	(*
			[1] ETA_3111U1006XHE321XXXXXXZ01, ELT_Zaehler_BHKW_321_01
			Primaer-Adresse = 1
			Seriennummer = 3999427
			[2] ETA_3111U1006XHE322XXXXXXZ01, ELT_Zaehler_BHKW_322_01
			Primaer-Adresse = 2
			Seriennummer = 3999432
			[3] ETA_3111U1006BEST001XXXXXXZ01, ELT_Zaehler_Buerotrakt_01
			Primaer-Adresse = 3
			Seriennummer = 120267
			[4] ETA_3111U1006BEST002XXXXXXZ01, ELT_Zaehler_Gebaede_01
			Primaer-Adresse = 4
			Seriennummer = 205684
			[5] ETA_3111U1006BEST003XXXXXXZ01, ELT_Zaehler_Halle_TGA_01
			Primaer-Adresse = 5
			Seriennummer = 120264
			[6] ETA_3111EG005BEST004XXXXXXZ01, ELT_Zaehler_Halle_Licht_01
			Primaer-Adresse = 6
			Seriennummer = 214516
			[7] ETA_3111U1006BEST007XXXXXXZ01, GAS_Zaehler BHKW_007_01
			Primaer-Adresse = 7
			Seriennummer = 42078747
			[8] ETA_3111U1006BEST008XXXXXXZ01, GAS_Zaehler BHKW_008_01
			Primaer-Adresse = 8
			Seriennummer = 42078748
			[9] ETA_3111U1006BEST071XXXXXXZ01, WAERME_Zaehler WP_945_4371_01
			Primaer-Adresse = 71
			Seriennummer = 67694371
			[10] ETA_3111U1006BEST072XXXXXXZ01, WAERME_Zaehler WP_945_4372_01
			Primaer-Adresse = 72
			Seriennummer = 67694372
	*)
	Kommunikation_MBus	: ST_MBUS_Communication;
	Komm_MBus_WZaehler	: ST_MBUS_Communication;
	Komm_MBus_WZaehler2	: ST_MBUS_Communication;
	Komm_MBus_WZaehler_Basement	: ST_MBUS_Communication;

	aTelegramm_WMZ350 						: ARRAY[1..cMBUS_MaxTelegrams] OF ST_MBus_Data2;
	aTelegramm_WMZ305 						: ARRAY[1..cMBUS_MaxTelegrams] OF ST_MBus_Data2;
	aTelegramm_WMZ100 						: ARRAY[1..cMBUS_MaxTelegrams] OF ST_MBus_Data2;
	aTelegramm_WMZ300 						: ARRAY[1..cMBUS_MaxTelegrams] OF ST_MBus_Data2;
	aTelegramm_WMZ245 						: ARRAY[1..cMBUS_MaxTelegrams] OF ST_MBus_Data2;
	aTelegramm_WMZ235 						: ARRAY[1..cMBUS_MaxTelegrams] OF ST_MBus_Data2;
	aTelegramm_WMZ405 						: ARRAY[1..cMBUS_MaxTelegrams] OF ST_MBus_Data2;
	aTelegramm_WMZ425 						: ARRAY[1..cMBUS_MaxTelegrams] OF ST_MBus_Data2;
	aTelegramm_WMZ455 						: ARRAY[1..cMBUS_MaxTelegrams] OF ST_MBus_Data2;
	aTelegramm_WMZ342 						: ARRAY[1..cMBUS_MaxTelegrams] OF ST_MBus_Data2;
	
	
	aTelegramm_WMZ900 						: ARRAY[1..cMBUS_MaxTelegrams] OF ST_MBus_Data2;
	aTelegramm_WMZ935 						: ARRAY[1..cMBUS_MaxTelegrams] OF ST_MBus_Data2;
	
	aTelegramm_WMZ135						: ARRAY[1..cMBUS_MaxTelegrams] OF ST_MBus_Data2;
	aTelegramm_WMZ138						: ARRAY[1..cMBUS_MaxTelegrams] OF ST_MBus_Data2;
	aTelegramm_WMZ105						: ARRAY[1..cMBUS_MaxTelegrams] OF ST_MBus_Data2;
	aTelegramm_WMZ710						: ARRAY[1..cMBUS_MaxTelegrams] OF ST_MBus_Data2;
	aTelegramm_WMZ205						: ARRAY[1..cMBUS_MaxTelegrams] OF ST_MBus_Data2;
	aTelegramm_WMZ720						: ARRAY[1..cMBUS_MaxTelegrams] OF ST_MBus_Data2;
	
	Telegramm_WZ_Brennwerttherme			: ARRAY[1..cMBUS_MaxTelegrams] OF ST_MBus_Data2;
	Telegramm_WZ_BHKW_1						: ARRAY[1..cMBUS_MaxTelegrams] OF ST_MBus_Data2;
	Telegramm_WZ_BHKW_2						: ARRAY[1..cMBUS_MaxTelegrams] OF ST_MBus_Data2;
	Telegramm_WZ_Druckluftkompressor		: ARRAY[1..cMBUS_MaxTelegrams] OF ST_MBus_Data2;
	Telegramm_WZ_PWT_1						: ARRAY[1..cMBUS_MaxTelegrams] OF ST_MBus_Data2;
	Telegramm_WZ_Ofenkuehlung				: ARRAY[1..cMBUS_MaxTelegrams] OF ST_MBus_Data2;
	Telegramm_WZ_Abwaerme_Ofen_Abgasfackel	: ARRAY[1..cMBUS_MaxTelegrams] OF ST_MBus_Data2;
	Telegramm_GZ331_BWT	: ARRAY[1..cMBUS_MaxTelegrams] OF ST_MBus_Data2;


	Telegramm_SZ_BHKW_321		: ARRAY[1..cMBUS_MaxTelegrams] OF ST_MBus_Data2;
	Telegramm_SZ_BHKW_322		: ARRAY[1..cMBUS_MaxTelegrams] OF ST_MBus_Data2;
	Telegramm_SZ_Buerotrakt		: ARRAY[1..cMBUS_MaxTelegrams] OF ST_MBus_Data2;
	Telegramm_SZ_Gebaeude		: ARRAY[1..cMBUS_MaxTelegrams] OF ST_MBus_Data2;
	Telegramm_SZ_Halle_TGA		: ARRAY[1..cMBUS_MaxTelegrams] OF ST_MBus_Data2;
	Telegramm_SZ_Halle_Licht	: ARRAY[1..cMBUS_MaxTelegrams] OF ST_MBus_Data2;

	Telegramm_GZ_BHKW_321		: ARRAY[1..cMBUS_MaxTelegrams] OF ST_MBus_Data2;
	Telegramm_GZ_BHKW_322		: ARRAY[1..cMBUS_MaxTelegrams] OF ST_MBus_Data2;

	Telegramm_WZ_4371_WP_946	: ARRAY[1..cMBUS_MaxTelegrams] OF ST_MBus_Data2;
	Telegramm_WZ_4372_WP_946	: ARRAY[1..cMBUS_MaxTelegrams] OF ST_MBus_Data2;
	
	maxNumberOfNodes :INT := 22;
	cMSRLIBMaxNumberOfMBusDevices : BYTE := 18;	(*~
				Maximale Anzahl an MBus Geräten, die von der MSRlib unterstützt werden.
				Diese Konstante wird auch für die DP-Historisierung verwendet und muss grösser 6 (Anzahl der Basisdatentypen) sein.
				*)
	cMBUS_MaxData : INT := 40;
	(*cMBUS_MaxTelegrams : INT := 2;
	cMBUS_MaxCom : INT := 1;*)

END_VAR

// ---- POUs/MBUS_WZaehler.TcPOU
PROGRAM MBUS_WZaehler (* hier wird die Klemme, an welche der M-Bus mit den Zählern angeschlossen ist, alle 10ms aufgerufen *)
VAR
	Komm_Klemme_WZaehler		: FB_MBUSKL6781;
	Komm_Klemme_WZaehler2		: FB_MBUSKL6781;

	
	WMZ331_Brennwerttherme				: FB_MBUS_General_Ext;	(*1*)
	WMZ321_BHKW_1						: FB_MBUS_General_Ext;	(*3*)
	WMZ322_BHKW_2						: FB_MBUS_General_Ext;	(*4*)
	WMZ251_Druckluftkompressor			: FB_MBUS_General_Ext;	(*5*)
	WMZ215_PWT_1						: FB_MBUS_General_Ext;	(*6*)
	WMZ261_Ofenkuehlung_Dichtungen		: FB_MBUS_General_Ext;	(*7*)
	WMZ361_Abwaerme_Ofen_Abgasfackel	: FB_MBUS_General_Ext;	(*8*)

	adrBrennwerttherme				: ST_MBus_SecAdr := (udiIdNumber:=16#00474907);
	adrBHKW_1						: ST_MBus_SecAdr := (udiIdNumber:=16#00470996);
	adrBHKW_2						: ST_MBus_SecAdr := (udiIdNumber:=16#00474904);
	adrDruckluftkompressor			: ST_MBus_SecAdr := (udiIdNumber:=16#00552639);
	adrPWT_1						: ST_MBus_SecAdr := (udiIdNumber:=16#00455395);
	adrOfenkuehlung_Dichtungen		: ST_MBus_SecAdr := (udiIdNumber:=16#00482160);
	adrAbwaerme_Ofen_Abgasfackel	: ST_MBus_SecAdr := (udiIdNumber:=16#00482192);

	

	
END_VAR

Komm_Klemme_WZaehler(stComIn := IN_WZaehler, stComOut := OUT_WZaehler, stCom := Komm_MBus_WZaehler); // FB_MBUSKL6781
WMZ331_Brennwerttherme(usiAddress := 253, stSecAdr := adrBrennwerttherme, stCom := Komm_MBus_WZaehler); // FB_MBUS_General_Ext
Telegramm_WZ_Brennwerttherme := WMZ331_Brennwerttherme.arrTelegram;
WMZ321_BHKW_1(usiAddress := 253, stSecAdr := adrBHKW_1, stCom := Komm_MBus_WZaehler); // FB_MBUS_General_Ext
Telegramm_WZ_BHKW_1 := WMZ321_BHKW_1.arrTelegram;
WMZ322_BHKW_2(usiAddress := 253, stSecAdr := adrBHKW_2, stCom := Komm_MBus_WZaehler); // FB_MBUS_General_Ext
WMZ251_Druckluftkompressor(
    usiAddress := 253,
    stSecAdr := adrDruckluftkompressor,
    stCom := Komm_MBus_WZaehler); // FB_MBUS_General_Ext
WMZ215_PWT_1(usiAddress := 253, stSecAdr := adrPWT_1, stCom := Komm_MBus_WZaehler); // FB_MBUS_General_Ext
WMZ261_Ofenkuehlung_Dichtungen(
    usiAddress := 253,
    stSecAdr := adrOfenkuehlung_Dichtungen,
    stCom := Komm_MBus_WZaehler); // FB_MBUS_General_Ext
Telegramm_WZ_Ofenkuehlung := WMZ261_Ofenkuehlung_Dichtungen.arrTelegram;
WMZ361_Abwaerme_Ofen_Abgasfackel(
    usiAddress := 253,
    stSecAdr := adrAbwaerme_Ofen_Abgasfackel,
    stCom := Komm_MBus_WZaehler); // FB_MBUS_General_Ext
Telegramm_WZ_Abwaerme_Ofen_Abgasfackel := WMZ361_Abwaerme_Ofen_Abgasfackel.arrTelegram;
Telegramm_WZ_BHKW_2 := WMZ322_BHKW_2.arrTelegram;
Telegramm_WZ_Druckluftkompressor := WMZ251_Druckluftkompressor.arrTelegram;
Telegramm_WZ_PWT_1 := WMZ215_PWT_1.arrTelegram;

END_PROGRAM

// ---- POUs/MBUS_WZaehler2.TcPOU
PROGRAM MBUS_WZaehler2 (* hier wird die Klemme, an welche der M-Bus mit den Zählern angeschlossen ist, alle 10ms aufgerufen *)
VAR
	Komm_Klemme_WZaehler2		: FB_MBUSKL6781;
	WMZ135						: FB_MBUS_General_Ext;
	WMZ138						: FB_MBUS_General_Ext;
	WMZ105						: FB_MBUS_General_Ext;
	WMZ710						: FB_MBUS_General_Ext;
	WMZ205						: FB_MBUS_General_Ext;
	WMZ720						: FB_MBUS_General_Ext;

	adrWMZ135			: ST_MBus_SecAdr := (udiIdNumber:=16#13859504);
	adrWMZ138			: ST_MBus_SecAdr := (udiIdNumber:=16#13859500);
	adrWMZ105			: ST_MBus_SecAdr := (udiIdNumber:=16#12675097);
	adrWMZ205			: ST_MBus_SecAdr := (udiIdNumber:=16#13859501);
	adrWMZ710			: ST_MBus_SecAdr := (udiIdNumber:=16#12675093);
	adrWMZ720			: ST_MBus_SecAdr := (udiIdNumber:=16#13859505);
END_VAR

WMZ138(usiAddress := 253, stSecAdr := adrWMZ138, stCom := Komm_MBus_WZaehler2); // FB_MBUS_General_Ext
Komm_Klemme_WZaehler2(stComIn := IN_WZaehler2, stComOut := OUT_WZaehler2, stCom := Komm_MBus_WZaehler2); // FB_MBUSKL6781
aTelegramm_WMZ138 := WMZ138.arrTelegram;
WMZ135(usiAddress := 253, stSecAdr := adrWMZ135, stCom := Komm_MBus_WZaehler2); // FB_MBUS_General_Ext
aTelegramm_WMZ135 := WMZ135.arrTelegram;
WMZ105(usiAddress := 253, stSecAdr := adrWMZ105, stCom := Komm_MBus_WZaehler2); // FB_MBUS_General_Ext
WMZ205(usiAddress := 253, stSecAdr := adrWMZ205, stCom := Komm_MBus_WZaehler2); // FB_MBUS_General_Ext
aTelegramm_WMZ105 := WMZ105.arrTelegram;
aTelegramm_WMZ205 := WMZ205.arrTelegram;
WMZ710(usiAddress := 253, stSecAdr := adrWMZ710, stCom := Komm_MBus_WZaehler2); // FB_MBUS_General_Ext
aTelegramm_WMZ710 := WMZ710.arrTelegram;
WMZ720(usiAddress := 253, stSecAdr := adrWMZ720, stCom := Komm_MBus_WZaehler2); // FB_MBUS_General_Ext
aTelegramm_WMZ720 := WMZ720.arrTelegram;

END_PROGRAM

// ---- POUs/MBUS_WZaehler_Basement.TcPOU
PROGRAM MBUS_WZaehler_Basement (* hier wird die Klemme, an welche der M-Bus mit den Zählern angeschlossen ist, alle 10ms aufgerufen *)
VAR
	Komm_Klemme_WZaehler_Basement 		: FB_MBUSKL6781;

	WMZ350								: FB_MBUS_General_Ext;
	WMZ305								: FB_MBUS_General_Ext;
	WMZ300								: FB_MBUS_General_Ext;
	WMZ100								: FB_MBUS_General_Ext;
	WMZ455								: FB_MBUS_General_Ext;
	WMZ245								: FB_MBUS_General_Ext;
	WMZ235								: FB_MBUS_General_Ext;
	WMZ425								: FB_MBUS_General_Ext;
	WMZ900								: FB_MBUS_General_Ext;
	WMZ935								: FB_MBUS_General_Ext;
	WMZ342								: FB_MBUS_General_Ext;
	WMZ405								: FB_MBUS_General_Ext;
	
	//basement
	adrWMZ350					: ST_MBus_SecAdr := (udiIdNumber:=16#75372672);
	adrWMZ305					: ST_MBus_SecAdr := (udiIdNumber:=16#75234689);
	adrWMZ100					: ST_MBus_SecAdr := (udiIdNumber:=16#75494412);
	adrWMZ300					: ST_MBus_SecAdr := (udiIdNumber:=16#75878308);
	
	adrWMZ455					: ST_MBus_SecAdr := (udiIdNumber:=16#75375855);
	adrWMZ245					: ST_MBus_SecAdr := (udiIdNumber:=16#75563317);
	adrWMZ235					: ST_MBus_SecAdr := (udiIdNumber:=16#13859503);
	adrWMZ425					: ST_MBus_SecAdr := (udiIdNumber:=16#75878305);
	adrWMZ900					: ST_MBus_SecAdr := (udiIdNumber:=16#72925041);
	adrWMZ935					: ST_MBus_SecAdr := (udiIdNumber:=16#72925042);
	adrWMZ342					: ST_MBus_SecAdr := (udiIdNumber:=16#75375999);
	adrWMZ405					: ST_MBus_SecAdr := (udiIdNumber:=16#76089225);

END_VAR

Komm_Klemme_WZaehler_Basement(
    stComIn := IN_WZaehler_Basement,
    stComOut := OUT_WZaehler_Basement,
    stCom := Komm_MBus_WZaehler_Basement); // FB_MBUSKL6781
WMZ350(usiAddress := 253, stSecAdr := adrWMZ350, stCom := Komm_MBus_WZaehler_Basement); // FB_MBUS_General_Ext
aTelegramm_WMZ350 := WMZ350.arrTelegram;
WMZ305(usiAddress := 253, stSecAdr := adrWMZ305, stCom := Komm_MBus_WZaehler_Basement); // FB_MBUS_General_Ext
aTelegramm_WMZ305 := WMZ305.arrTelegram;
WMZ100(usiAddress := 253, stSecAdr := adrWMZ100, stCom := Komm_MBus_WZaehler_Basement); // FB_MBUS_General_Ext
WMZ300(usiAddress := 253, stSecAdr := adrWMZ300, stCom := Komm_MBus_WZaehler_Basement); // FB_MBUS_General_Ext
aTelegramm_WMZ100 := WMZ100.arrTelegram;
aTelegramm_WMZ300 := WMZ300.arrTelegram;
WMZ455(usiAddress := 253, stSecAdr := adrWMZ455, stCom := Komm_MBus_WZaehler_Basement); // FB_MBUS_General_Ext
aTelegramm_WMZ455 := WMZ455.arrTelegram;
WMZ245(usiAddress := 253, stSecAdr := adrWMZ245, stCom := Komm_MBus_WZaehler_Basement); // FB_MBUS_General_Ext
aTelegramm_WMZ245 := WMZ245.arrTelegram;
WMZ235(usiAddress := 253, stSecAdr := adrWMZ235, stCom := Komm_MBus_WZaehler_Basement); // FB_MBUS_General_Ext
aTelegramm_WMZ235 := WMZ235.arrTelegram;
WMZ425(usiAddress := 253, stSecAdr := adrWMZ425, stCom := Komm_MBus_WZaehler_Basement); // FB_MBUS_General_Ext
aTelegramm_WMZ425 := WMZ425.arrTelegram;
WMZ900(usiAddress := 253, stSecAdr := adrWMZ900, stCom := Komm_MBus_WZaehler_Basement); // FB_MBUS_General_Ext
aTelegramm_WMZ900 := WMZ900.arrTelegram;
WMZ935(usiAddress := 253, stSecAdr := adrWMZ935, stCom := Komm_MBus_WZaehler_Basement); // FB_MBUS_General_Ext
aTelegramm_WMZ935 := WMZ935.arrTelegram;
WMZ342(usiAddress := 253, stSecAdr := adrWMZ342, stCom := Komm_MBus_WZaehler_Basement); // FB_MBUS_General_Ext
aTelegramm_WMZ342 := WMZ342.arrTelegram;
WMZ405(usiAddress := 253, stSecAdr := adrWMZ405, stCom := Komm_MBus_WZaehler_Basement); // FB_MBUS_General_Ext
aTelegramm_WMZ405 := WMZ405.arrTelegram;

END_PROGRAM

// ---- POUs/MBUS_Zaehler.TcPOU
PROGRAM MBUS_Zaehler (* hier wird die Klemme, an welche der M-Bus mit den Zählern angeschlossen ist, alle 10ms aufgerufen *)
VAR
	Kommunikation_Klemme: FB_MBUSKL6781;

	Stromzaehler_BHKW_321		: FB_MBUS_General_Ext;
	Stromzaehler_BHKW_322	: FB_MBUS_General_Ext;
	Stromzaehler_Buerotrakt	: FB_MBUS_General_Ext;

	Stromzaehler_Gebaeude: FB_MBUS_General_Ext;
	Stromzaehler_Halle_TGA: FB_MBUS_General_Ext;
	Stromzaehler_Halle_Licht: FB_MBUS_General_Ext;
	Gaszaehler_BHKW1: FB_MBUS_General_Ext;
	Gaszaehler_BHKW2: FB_MBUS_General_Ext;

	WZ_4371_WP_946	: FB_MBUS_General_Ext;
	WZ_4372_WP_946	: FB_MBUS_General_Ext;
	
	
	
	
	
END_VAR

Kommunikation_Klemme(stComIn := IN_Stromzaehler, stComOut := OUT_Stromzaehler, stCom := Kommunikation_MBus); // FB_MBUSKL6781
Stromzaehler_BHKW_321(usiAddress := 1, stCom := Kommunikation_MBUS); // FB_MBUS_General_Ext
Telegramm_SZ_BHKW_321 := Stromzaehler_BHKW_321.arrTelegram;
Stromzaehler_BHKW_322(usiAddress := 2, stCom := Kommunikation_MBUS); // FB_MBUS_General_Ext
Telegramm_SZ_BHKW_322 := Stromzaehler_BHKW_322.arrTelegram;
Stromzaehler_Buerotrakt(usiAddress := 3, stCom := Kommunikation_MBUS); // FB_MBUS_General_Ext
Stromzaehler_Gebaeude(usiAddress := 4, stCom := Kommunikation_MBUS); // FB_MBUS_General_Ext
Stromzaehler_Halle_TGA(usiAddress := 5, stCom := Kommunikation_MBUS); // FB_MBUS_General_Ext
Stromzaehler_Halle_Licht(usiAddress := 6, stCom := Kommunikation_MBUS); // FB_MBUS_General_Ext
Telegramm_SZ_Halle_Licht := Stromzaehler_Halle_Licht.arrTelegram;
Gaszaehler_BHKW1(usiAddress := 7, stCom := Kommunikation_MBUS); // FB_MBUS_General_Ext
Telegramm_GZ_BHKW_321 := Gaszaehler_BHKW1.arrTelegram;
Gaszaehler_BHKW2(usiAddress := 8, stCom := Kommunikation_MBUS); // FB_MBUS_General_Ext
Telegramm_SZ_Buerotrakt := Stromzaehler_Buerotrakt.arrTelegram;
Telegramm_SZ_Gebaeude := Stromzaehler_Gebaeude.arrTelegram;
Telegramm_SZ_Halle_TGA := Stromzaehler_Halle_TGA.arrTelegram;
Telegramm_GZ_BHKW_322 := Gaszaehler_BHKW2.arrTelegram;
WZ_4371_WP_946(usiAddress := 71, stCom := Kommunikation_MBUS); // FB_MBUS_General_Ext
Telegramm_WZ_4371_WP_946 := WZ_4371_WP_946.arrTelegram;
WZ_4372_WP_946(usiAddress := 72, stCom := Kommunikation_MBUS); // FB_MBUS_General_Ext
Telegramm_WZ_4372_WP_946 := WZ_4372_WP_946.arrTelegram;

END_PROGRAM

// ---- POUs/MAIN.TcPOU
PROGRAM MAIN
VAR
	init_done		: BOOL := FALSE;
	
	//strategy controller
	Strategy : FB_StrategyController;
	//Strategy : FB_StrategyController_noChiller;
	//Strategy : FB_Strategycontroller_Conventional;
	//Strategy : FB_Strategycontroller_NoStorages;
	
	//thermal networks
	CN : FB_CoolingNetwork;
	HNLT_CN : FB_HnltCnLinkage;
	HNHT_CN : FB_HnhtCnLinkage;
	HNLT : FB_HeatingNetworkLowTemperature;
	HNHT_HNLT : FB_HnhtHnltLinkage;
	HNHT : FB_HeatingNetworkHighTemperature;

	
	//ambient state
	Ambient : FB_Ambient;
	
	//sensors
	LowVoltageMainDistribution : FB_LowVoltageMainDistribution;
END_VAR

//strategy controller
Strategy(ambientState := Ambient.localState,
	cnState := CN.localState,
	hnltState := HNLT.localState,
	hnhtState := HNHT.localState);

//ambient state
Ambient(sIPAddress := GlobalVariables.sIP_Ventilation);

//sensors
LowVoltageMainDistribution();
	
//thermal networks
CN(controlAutomatic := Strategy.cnControl);

HNLT_CN(controlAutomatic := Strategy.hnltCnLinkageControl,
	stAmbientState := Ambient.localState);
	
HNHT_CN(controlAutomatic := Strategy.hnhtCnLinkageControl);
	
HNLT(ambientState := Ambient.localState,
	controlAutomatic := Strategy.hnltControl);
	
HNHT_HNLT(controlAutomatic := Strategy.hnhtHnltLinkageControl);
	
HNHT(controlAutomatic := Strategy.hnhtControl,
	stAmbientState := Ambient.localState);
	


//Current implementation

(* --------------------------------------------------------------------------------------------------------------------------- *)

(* Analog- & Binaer Eingaenge - LESEN *)
(* P_Lesen; *)

	(* BUS Kommunikation - LESEN *)

(* --------------------------------------------------------------------------------------------------------------------------- *)
(* Starte Sub-Applikationen *)


	(*Initialisierung des Systems*)
	(*Einmalige Initialisierung der Parameter bei Hochlauf*)
	IF(NOT init_done) THEN
		Initialisierungsroutine();
		init_done := TRUE;
	END_IF;

	(* Allgemeine Parameter (Systemszeit, usw.) *)
	GA_Allgemein();

	(* Beleuchtung *)
	Beleuchtung();

END_PROGRAM

// ---- POUs/06 Strategy/FB_StrategyController.TcPOU
FUNCTION_BLOCK FB_StrategyController
VAR_INPUT
	ambientState : ST_AmbientState;
	
	//actual temperatures in thermal networks
	cnState : ST_ThermalNetworkState;
	hnltState : ST_ThermalNetworkState;
	hnhtState : ST_ThermalNetworkState;
END_VAR
VAR_OUTPUT	
	cnControl : ST_CoolingNetworkControl;
	hnltControl : ST_HeatingNetworkLowTemperatureControl;	
	hnhtControl : ST_HeatingNetworkHighTemperatureControl;
	hnltCnLinkageControl : ST_HnltCnLinkageControl;
	hnhtHnltLinkageControl : ST_HnhtHnltLinkageControl;
	hnhtCnLinkageControl : ST_HnhtCnLinkageControl;
END_VAR
VAR
	{attribute 'OPC.UA.DA' := '1'}
	localSetParameters : ST_StrategySetParameters;	
	{attribute 'OPC.UA.DA' := '1'}
	localState : ST_StrategyState;	

	//default parameters
	localDefaultParameters : ST_StrategyDefaultParameters;

	//internal variables
	fTargetTemperature_HNHT_Heating : REAL;
	fTargetTemperature_HNHT_Cooling : REAL;
	fTargetTemperature_HNLT_Cooling : REAL;
	fTargetTemperature_HNLT_Heating : REAL;
	fTargetTemperature_CN : REAL;
	aTemperatureLimits_HNHT : ARRAY[1..2] OF REAL;
	aTemperatureLimits_HNLT : ARRAY[1..2] OF REAL;
	aTemperatureLimits_CN : ARRAY[1..2] OF REAL;
	stHNHTCheckDefaultParameters : ST_RangeCheckDefaultParameters := (tTaskCycleTime := GlobalVariables.tCtrlCycleTime_MAIN, tCtrlCycleTime := GlobalVariables.tCtrlCycleTime_MAIN, fRestoreDifference := 5);
	HNHT_Check : FB_RangeCheck := (ST_DefaultParameters := stHNHTCheckDefaultParameters);
	stHNLTCheckDefaultParameters : ST_RangeCheckDefaultParameters := (tTaskCycleTime := GlobalVariables.tCtrlCycleTime_MAIN, tCtrlCycleTime := GlobalVariables.tCtrlCycleTime_MAIN, fRestoreDifference := 5);
	HNLT_Check : FB_RangeCheck := (ST_DefaultParameters := stHNLTCheckDefaultParameters);
	stCNCheckDefaultParameters : ST_RangeCheckDefaultParameters := (tTaskCycleTime := GlobalVariables.tCtrlCycleTime_MAIN, tCtrlCycleTime := GlobalVariables.tCtrlCycleTime_MAIN, fRestoreDifference := 2);
	CN_Check : FB_RangeCheck := (ST_DefaultParameters := stCNCheckDefaultParameters);
	
	
	//controller and variables for high temperature heating network
	fOffset_TargetTemperature_CHP1 : REAL; //not fixed, switches depending on ambient temperature -> see method: ControlHNHT
	fOffset_TargetTemperature_CHP2 : REAL; //not fixed, switches depending on ambient temperature -> see method: ControlHNHT
	fOffset_TargetTemperature_CondensingBoiler : REAL := 2;
	Controller_CHP_Prioritization : FB_CTRL_2POINT;
	Controller_CHP_Prioritization_Parameters : ST_CTRL_2POINT_PARAMS;	
	Controller_CHP1_UpperTemperature : FB_CTRL_2POINT; //check upper temperature for turning on chp
	Controller_CHP1_LowerTemperature : FB_CTRL_2POINT; //check lower temperature for turning off chp
	Controller_CHP1_Parameters : ST_CTRL_2POINT_PARAMS;	
	Trigger_CHP1_UpperTemperature : F_TRIG;
	Trigger_CHP1_LowerTemperature : F_TRIG;
	bTrigger_CHP1 : BOOL;
	Controller_CHP2_UpperTemperature : FB_CTRL_2POINT;
	Controller_CHP2_LowerTemperature : FB_CTRL_2POINT;
	Controller_CHP2_Parameters : ST_CTRL_2POINT_PARAMS;
	Trigger_CHP2_UpperTemperature : F_TRIG;
	Trigger_CHP2_LowerTemperature : F_TRIG;
	bTrigger_CHP2 : BOOL;
	Controller_CondensingBoiler : FB_CTRL_2POINT;
	Controller_CondensingBoiler_Parameters : ST_CTRL_2POINT_PARAMS;
	Controller_VSI_Loading_Permission : FB_CTRL_2POINT;
	Controller_VSI_Loading_Permission_Parameters : ST_CTRL_2POINT_PARAMS;
	Controller_VSI_Unloading_Permission : FB_CTRL_2POINT;
	Controller_VSI_Unloading_Permission_Parameters : ST_CTRL_2POINT_PARAMS;
	Controller_Buffer_VSI_Unloading : FB_CTRL_2POINT;
	Controller_Buffer_VSI_Unloading_Parameters : ST_CTRL_2POINT_PARAMS;
	Controller_StaticHeating : FB_CTRL_2POINT;
	Controller_StaticHeating_Parameters : ST_CTRL_2POINT_PARAMS;
	
	//controllers and variables for low temperature heating network
	Controller_OuterCapillaryTubeMats : FB_CTRL_2POINT;
	Controller_OuterCapillaryTubeMats_Parameters : ST_CTRL_2POINT_PARAMS;
	Controller_OuterCapillaryTubeMats_Permission : FB_CTRL_2POINT;
	Controller_OuterCapillaryTubeMats_Permission_Parameters : ST_CTRL_2POINT_PARAMS;
	fOffset_TargetTemperature_OuterCapillaryTubeMats_Cooling : REAL := 1;	
	fOffset_OuterCapillaryTubeMats_Permission : REAL := 10;
	
	Controller_HVFA_HNLT_HVFALoadingPermission : FB_CTRL_2POINT;
	Controller_HVFA_HNLT_HVFALoadingPermission_Parameters : ST_CTRL_2POINT_PARAMS;
	Controller_HVFA_HNLT_HVFAUnloadingPermission : FB_CTRL_2POINT;
	Controller_HVFA_HNLT_HVFAUnloadingPermission_Parameters : ST_CTRL_2POINT_PARAMS;
	Controller_Buffer_HVFA_HNLT_HVFAUnloading : FB_CTRL_2POINT;
	Controller_Buffer_HVFA_HNLT_HVFAUnloading_Parameters : ST_CTRL_2POINT_PARAMS;
	Controller_Buffer_HVFA_HNLT_HVFALoading : FB_CTRL_2POINT;
	Controller_Buffer_HVFA_HNLT_HVFALoading_Parameters : ST_CTRL_2POINT_PARAMS;
	Controller_HVFA_HNLT_Recooling : FB_CTRL_2POINT;
	Controller_HVFA_HNLT_Recooling_Parameters : ST_CTRL_2POINT_PARAMS;
	fOffset_TargetTemperature_HVFA_HNLT_Heating : REAL := 1;
	fOffset_HVFA_HNLT_Recooling : REAL := 16;
	fOffset_HVFA_HNLT_HVFALoadingPermission : REAL := 6;
	fOffset_Buffer_HVFA_HNLT_HVFALoading : REAL := 2;
		
	
	//controllers and variables for cooling network
	fOffset_TargetTemperature_eChiller : REAL := 2;	
	fOffset_TargetTemperature_HVFA_CN : REAL := 1;
	fOffset_TargetTemperature_HVFA_CN_Permission : REAL := 2.5;
	Controller_eChiller : FB_CTRL_2POINT;
	Controller_eChiller_Parameters : ST_CTRL_2POINT_PARAMS;	
	Controller_HVFA_CN_UnloadingPermission : FB_CTRL_2POINT;
	Controller_HVFA_CN_UnloadingPermission_Parameters : ST_CTRL_2POINT_PARAMS;
	Controller_Buffer_HVFA_CN_Unloading : FB_CTRL_2POINT;
	Controller_Buffer_HVFA_CN_Unloading_Parameters : ST_CTRL_2POINT_PARAMS;

	//controllers and variables for hnht and hnlt linkage
	Controller_HeatExchanger1 : FB_CTRL_2POINT;
	Controller_HeatExchanger1_Parameters : ST_CTRL_2POINT_PARAMS;
	fOffset_TargetTemperature_HeatExchanger1 : REAL := 2;
	Controller_HeatPump_HNHT : FB_CTRL_2POINT;
	Controller_HeatPump_HNHT_Parameters : ST_CTRL_2POINT_PARAMS;
	fOffset_TargetTemperature_HeatPump_HNHT : REAL := 3;
	Controller_HeatPump_HNLT : FB_CTRL_2POINT;
	Controller_HeatPump_HNLT_Parameters : ST_CTRL_2POINT_PARAMS;
	fOffset_TargetTemperature_HeatPump_HNHT_Permission : REAL := 4;
	
	//controllers and variables for hnlt and cn linkage
	fOffset_TargetTemperature_HeatPump : REAL;
	fOffset_TargetTemperature_HeatPump_Lower_CN_Permission : REAL;
	fOffset_TargetTemperature_HeatPump_Upper_CN_Permission : REAL;
	Controller_HeatPump : FB_CTRL_2POINT;
	Controller_HeatPump_Parameters : ST_CTRL_2POINT_PARAMS;
	Controller_HeatPump_Permission_Upper_CN : FB_CTRL_2POINT;
	Controller_HeatPump_Permission_Upper_CN_Parameters : ST_CTRL_2POINT_PARAMS;		
	Controller_HeatPump_Permission_Lower_CN : FB_CTRL_2POINT;
	Controller_HeatPump_Permission_Lower_CN_Parameters : ST_CTRL_2POINT_PARAMS;	

	//clock
	stDefaultParameters_Clock : ST_ClockDefaultParameters := (tTaskCycleTime := GlobalVariables.tCtrlCycleTime_MAIN, tCtrlCycleTime := T#1M);
	Clock : FB_Clock := (ST_DefaultParameters := stDefaultParameters_Clock);
END_VAR

Clock();
AmbientControl();
SetTemperatures();
ControlCN();
ControlHNLT();
ControlHNHT();
ControlHnltCnLinkage();
ControlHnhtHnltLinkage();
SetState();

METHOD AmbientControl : BOOL
VAR_INPUT
END_VAR
//check for heating or cooling mode
IF Clock.stClockState.sintMonth>4 AND Clock.stClockState.sintMonth<9 THEN
	//heating mode
	hnltCnLinkageControl.bHeatingMode := FALSE;
	hnhtCnLinkageControl.bHeatingMode := FALSE;
	localState.bHeatingMode := FALSE;
ELSE
	//cooling mode	
	hnltCnLinkageControl.bHeatingMode := TRUE;
	hnhtCnLinkageControl.bHeatingMode := TRUE;
	localState.bHeatingMode := TRUE;
END_IF
END_METHOD

METHOD ControlCN : BOOL
VAR_INPUT
END_VAR
//set hysteresis parameters for two-point controllers in cooling network
Controller_eChiller_Parameters.fHysteresisRange := 4;
Controller_eChiller_Parameters.tCtrlCycleTime := GlobalVariables.tCtrlCycleTime_MAIN;
Controller_eChiller_Parameters.tTaskCycleTime := GlobalVariables.tTaskCycleTime_MAIN;

//permission to unload storage depending on upper hvfa storage temperature
Controller_HVFA_CN_UnloadingPermission_Parameters.fHysteresisRange := 1;
Controller_HVFA_CN_UnloadingPermission_Parameters.tCtrlCycleTime := GlobalVariables.tCtrlCycleTime_MAIN;
Controller_HVFA_CN_UnloadingPermission_Parameters.tTaskCycleTime := GlobalVariables.tTaskCycleTime_MAIN;

//hysteresis for unloading hvfa storage depending on buffer storage temperature
Controller_Buffer_HVFA_CN_Unloading_Parameters.fHysteresisRange := 2;
Controller_Buffer_HVFA_CN_Unloading_Parameters.tCtrlCycleTime := GlobalVariables.tCtrlCycleTime_MAIN;
Controller_Buffer_HVFA_CN_Unloading_Parameters.tTaskCycleTime := GlobalVariables.tTaskCycleTime_MAIN;

//control eChiller
Controller_eChiller(fSetpointValue := cnState.fMidTemperature,
	fActualValue := fTargetTemperature_CN+fOffset_TargetTemperature_eChiller,
	eMode := eCTRL_MODE_ACTIVE,
	stParams := Controller_eChiller_Parameters);
	
//control hvfa storage unloading permission 
Controller_HVFA_CN_UnloadingPermission(fSetpointValue := fTargetTemperature_CN-fOffset_TargetTemperature_HVFA_CN_Permission,
	fActualValue := cnState.fLowerTemperature_ActiveStorage,
	eMode := eCTRL_MODE_ACTIVE,
	stParams := Controller_HVFA_CN_UnloadingPermission_Parameters);
	
//unloading permission buffer HVFA
Controller_Buffer_HVFA_CN_Unloading(fSetpointValue := cnState.fMidTemperature,
	fActualValue := fTargetTemperature_CN+fOffset_TargetTemperature_HVFA_CN,
	eMode := eCTRL_MODE_ACTIVE,
	stParams := Controller_Buffer_HVFA_CN_Unloading_Parameters);
	
//cnControl.bSetStatusOn_eChiller := Controller_eChiller.bOut;
//cnControl.bSetStatusOn_HVFASystem := (Controller_Buffer_HVFA_CN_Unloading.bOut AND Controller_HVFA_CN_UnloadingPermission.bOut) OR (hnltCnLinkageControl.bSetStatusOn_HeatPump AND NOT Controller_Buffer_HVFA_CN_Unloading.bOut AND NOT Controller_HVFA_CN_UnloadingPermission.bOut); 
//cnControl.bLoading_HVFASystem := NOT (Controller_Buffer_HVFA_CN_Unloading.bOut AND Controller_HVFA_CN_UnloadingPermission.bOut);

cnControl.bSetStatusOn_eChiller := TRUE;
cnControl.bSetStatusOn_HVFASystem := FALSE;
cnControl.bLoading_HVFASystem := FALSE;
END_METHOD

METHOD ControlHNHT : BOOL
VAR_INPUT
END_VAR
VAR
END_VAR
//set hysteresis parameters for two-point controllers in high temperature heating network
Controller_CHP_Prioritization_Parameters.fHysteresisRange := 4;
Controller_CHP_Prioritization_Parameters.tCtrlCycleTime := GlobalVariables.tCtrlCycleTime_MAIN;
Controller_CHP_Prioritization_Parameters.tTaskCycleTime := GlobalVariables.tTaskCycleTime_MAIN;

Controller_CHP1_Parameters.tCtrlCycleTime := GlobalVariables.tCtrlCycleTime_MAIN;
Controller_CHP1_Parameters.tTaskCycleTime := GlobalVariables.tTaskCycleTime_MAIN;
Controller_CHP2_Parameters.tCtrlCycleTime := GlobalVariables.tCtrlCycleTime_MAIN;
Controller_CHP2_Parameters.tTaskCycleTime := GlobalVariables.tTaskCycleTime_MAIN;

Controller_CondensingBoiler_Parameters.fHysteresisRange := 8;
Controller_CondensingBoiler_Parameters.tCtrlCycleTime := GlobalVariables.tCtrlCycleTime_MAIN;
Controller_CondensingBoiler_Parameters.tTaskCycleTime := GlobalVariables.tTaskCycleTime_MAIN;

Controller_Buffer_VSI_Unloading_Parameters.fHysteresisRange := 4;
Controller_Buffer_VSI_Unloading_Parameters.tCtrlCycleTime := GlobalVariables.tCtrlCycleTime_MAIN;
Controller_Buffer_VSI_Unloading_Parameters.tTaskCycleTime := GlobalVariables.tTaskCycleTime_MAIN;

Controller_VSI_Unloading_Permission_Parameters.fHysteresisRange := 4;
Controller_VSI_Unloading_Permission_Parameters.tCtrlCycleTime := GlobalVariables.tCtrlCycleTime_MAIN;
Controller_VSI_Unloading_Permission_Parameters.tTaskCycleTime := GlobalVariables.tTaskCycleTime_MAIN;

Controller_VSI_Loading_Permission_Parameters.fHysteresisRange := 4;
Controller_VSI_Loading_Permission_Parameters.tCtrlCycleTime := GlobalVariables.tCtrlCycleTime_MAIN;
Controller_VSI_Loading_Permission_Parameters.tTaskCycleTime := GlobalVariables.tTaskCycleTime_MAIN;

Controller_StaticHeating_Parameters.fHysteresisRange := 4;
Controller_StaticHeating_Parameters.tCtrlCycleTime := GlobalVariables.tCtrlCycleTime_MAIN;
Controller_StaticHeating_Parameters.tTaskCycleTime := GlobalVariables.tTaskCycleTime_MAIN;

Controller_CHP_Prioritization(fSetpointValue := 15,
	fActualValue := ambientState.fOutsideTemperature_Mean,
	eMode := eCTRL_MODE_ACTIVE,
	stParams := Controller_CHP_Prioritization_Parameters);
IF Controller_CHP_Prioritization.bOut THEN
	//prioritize large CHP (CHP2) during cold temperatures
	Controller_CHP1_Parameters.fHysteresisRange := 14;
	Controller_CHP2_Parameters.fHysteresisRange := 12;
	fOffset_TargetTemperature_CHP1 := 1;
	fOffset_TargetTemperature_CHP2 := 0;
ELSE
	//prioritize large CHP (CHP2) during cold temperatures
	Controller_CHP1_Parameters.fHysteresisRange := 12;
	Controller_CHP2_Parameters.fHysteresisRange := 14;	
	fOffset_TargetTemperature_CHP1 := 0;
	fOffset_TargetTemperature_CHP2 := 1;	
END_IF

//start when upper temperature too cold and stop when lower temperature too hot
Controller_CHP1_UpperTemperature(fSetpointValue := fTargetTemperature_HNHT_Heating-fOffset_TargetTemperature_CHP1,
	fActualValue := hnhtState.fUpperTemperature,
	eMode := eCTRL_MODE_ACTIVE,
	stParams := Controller_CHP1_Parameters);
Controller_CHP1_LowerTemperature(fSetpointValue := fTargetTemperature_HNHT_Heating-fOffset_TargetTemperature_CHP1,
	fActualValue := hnhtState.fLowerTemperature,
	eMode := eCTRL_MODE_ACTIVE,
	stParams := Controller_CHP1_Parameters);
Trigger_CHP1_UpperTemperature(CLK := Controller_CHP1_UpperTemperature.bOut);
Trigger_CHP1_LowerTemperature(CLK := Controller_CHP1_LowerTemperature.bOut);
IF Trigger_CHP1_UpperTemperature.Q THEN
	bTrigger_CHP1 := TRUE;
END_IF
IF Trigger_CHP1_LowerTemperature.Q THEN
	bTrigger_CHP1 := FALSE;
END_IF
hnhtControl.bSetStatusOn_CHP1 := Controller_CHP1_UpperTemperature.bOut OR (Controller_CHP1_LowerTemperature.bOut AND bTrigger_CHP1);

//start when upper temperature too cold and stop when lower temperature too hot
Controller_CHP2_UpperTemperature(fSetpointValue := fTargetTemperature_HNHT_Heating-fOffset_TargetTemperature_CHP2,
	fActualValue := hnhtState.fUpperTemperature,
	eMode := eCTRL_MODE_ACTIVE,
	stParams := Controller_CHP2_Parameters);
Controller_CHP2_LowerTemperature(fSetpointValue := fTargetTemperature_HNHT_Heating-fOffset_TargetTemperature_CHP2,
	fActualValue := hnhtState.fLowerTemperature,
	eMode := eCTRL_MODE_ACTIVE,
	stParams := Controller_CHP2_Parameters);
Trigger_CHP2_UpperTemperature(CLK := Controller_CHP2_UpperTemperature.bOut);
Trigger_CHP2_LowerTemperature(CLK := Controller_CHP2_LowerTemperature.bOut);
IF Trigger_CHP2_UpperTemperature.Q THEN
	bTrigger_CHP2 := TRUE;
END_IF
IF Trigger_CHP2_LowerTemperature.Q THEN
	bTrigger_CHP2 := FALSE;
END_IF
hnhtControl.bSetStatusOn_CHP2 := Controller_CHP2_UpperTemperature.bOut OR (Controller_CHP2_LowerTemperature.bOut AND bTrigger_CHP2);

Controller_CondensingBoiler(fSetpointValue := fTargetTemperature_HNHT_Heating-fOffset_TargetTemperature_CondensingBoiler,
	fActualValue := hnhtState.fMidTemperature,
	eMode := eCTRL_MODE_ACTIVE,
	stParams := Controller_CondensingBoiler_Parameters);
hnhtControl.bSetStatusOn_CondensingBoiler := Controller_CondensingBoiler.bOut;

//buffer storage asks VSI for unloading when buffer storage temperature falls below limit
Controller_Buffer_VSI_Unloading(fSetpointValue := fTargetTemperature_HNHT_Heating,
	fActualValue := hnhtState.fMidTemperature,
	eMode := eCTRL_MODE_ACTIVE,
	stParams := Controller_Buffer_VSI_Unloading_Parameters);

//VSI storage may only be unloaded when upper temperature is between limits for unloading
Controller_VSI_Unloading_Permission(fSetpointValue := hnhtState.fUpperTemperature_ActiveStorage,
	fActualValue := fTargetTemperature_HNHT_Heating,
	eMode := eCTRL_MODE_ACTIVE,
	stParams := Controller_VSI_Unloading_Permission_Parameters);
	
//VSI storage may only be loaded when lower temperature is between limits for loading
Controller_VSI_Loading_Permission(fSetpointValue := fTargetTemperature_HNHT_Heating,
	fActualValue := hnhtState.fLowerTemperature_ActiveStorage,
	eMode := eCTRL_MODE_ACTIVE,
	stParams := Controller_VSI_Loading_Permission_Parameters);
	
hnhtControl.bSetStatusOn_VSIStorage := (Controller_Buffer_VSI_Unloading.bOut AND Controller_VSI_Unloading_Permission.bOut AND NOT (hnhtControl.bSetStatusOn_CHP1 OR hnhtControl.bSetStatusOn_CHP2)) OR ((hnhtControl.bSetStatusOn_CHP1 OR hnhtControl.bSetStatusOn_CHP2) AND NOT Controller_Buffer_VSI_Unloading.bOut AND Controller_VSI_Loading_Permission.bOut); 
hnhtControl.bLoading_VSISystem := NOT Controller_Buffer_VSI_Unloading.bOut;

//condensing boiler is switched if network temperature falls below critical temperature limit
Controller_StaticHeating(fSetpointValue := 15,
	fActualValue := ambientState.fOutsideTemperature,
	eMode := eCTRL_MODE_ACTIVE,
	stParams := Controller_StaticHeating_Parameters);
hnhtControl.bSetStatusOn_StaticHeating := Controller_StaticHeating.bOut;
END_METHOD

METHOD ControlHnhtHnltLinkage : BOOL
VAR_INPUT
END_VAR
Controller_HeatExchanger1_Parameters.fHysteresisRange := 8;
Controller_HeatExchanger1_Parameters.tCtrlCycleTime := GlobalVariables.tCtrlCycleTime_MAIN;
Controller_HeatExchanger1_Parameters.tTaskCycleTime := GlobalVariables.tTaskCycleTime_MAIN;

Controller_HeatPump_HNHT_Parameters.fHysteresisRange := 4;
Controller_HeatPump_HNHT_Parameters.tCtrlCycleTime := GlobalVariables.tCtrlCycleTime_MAIN;
Controller_HeatPump_HNHT_Parameters.tTaskCycleTime := GlobalVariables.tTaskCycleTime_MAIN;

Controller_HeatPump_HNLT_Parameters.fHysteresisRange := 4;
Controller_HeatPump_HNLT_Parameters.tCtrlCycleTime := GlobalVariables.tCtrlCycleTime_MAIN;
Controller_HeatPump_HNLT_Parameters.tTaskCycleTime := GlobalVariables.tTaskCycleTime_MAIN;

//control heat exchanger 1
Controller_HeatExchanger1(fSetpointValue := fTargetTemperature_HNLT_Heating-fOffset_TargetTemperature_HeatExchanger1,
	fActualValue := hnltState.fMidTemperature,
	eMode := eCTRL_MODE_ACTIVE,
	stParams := Controller_HeatExchanger1_Parameters);
hnhtHnltLinkageControl.bSetStatusOn_HeatExchanger1 := Controller_HeatExchanger1.bOut;

//control heat pump hnht, return temperature HNHT should not exceed 60 °C
Controller_HeatPump_HNHT(fSetpointValue := fTargetTemperature_HNHT_Heating+fOffset_TargetTemperature_HeatPump_HNHT,
	fActualValue := hnhtState.fLowerTemperature,
	eMode := eCTRL_MODE_ACTIVE,
	stParams := Controller_HeatPump_HNHT_Parameters);
	
Controller_HeatPump_HNLT(fSetpointValue := hnltState.fMidTemperature,
	fActualValue := fTargetTemperature_HNLT_Cooling-fOffset_TargetTemperature_HeatPump_HNHT_Permission,
	eMode := eCTRL_MODE_ACTIVE,
	stParams := Controller_HeatPump_HNLT_Parameters);	
	
// If requested to cool HNLT and HNHT is not too hot, activate heat pump
hnhtHnltLinkageControl.bSetStatusOn_HeatPump := Controller_HeatPump_HNHT.bOut AND Controller_HeatPump_HNLT.bOut;
END_METHOD

METHOD ControlHNLT : BOOL
VAR_INPUT
END_VAR
//set hysteresis parameters for two-point controllers in cooling network
Controller_OuterCapillaryTubeMats_Parameters.fHysteresisRange := 6;
Controller_OuterCapillaryTubeMats_Parameters.tCtrlCycleTime := GlobalVariables.tCtrlCycleTime_MAIN;
Controller_OuterCapillaryTubeMats_Parameters.tTaskCycleTime := GlobalVariables.tTaskCycleTime_MAIN;

Controller_OuterCapillaryTubeMats_Permission_Parameters.fHysteresisRange := 6;
Controller_OuterCapillaryTubeMats_Permission_Parameters.tCtrlCycleTime := GlobalVariables.tCtrlCycleTime_MAIN;
Controller_OuterCapillaryTubeMats_Permission_Parameters.tTaskCycleTime := GlobalVariables.tTaskCycleTime_MAIN;


//control strategy for cooling network - fSetpointValue and fActualValue are changed for cooling applications
Controller_OuterCapillaryTubeMats(fSetpointValue := hnltState.fMidTemperature,
	fActualValue := fTargetTemperature_HNLT_Cooling+fOffset_TargetTemperature_OuterCapillaryTubeMats_Cooling,
	eMode := eCTRL_MODE_ACTIVE,
	stParams := Controller_OuterCapillaryTubeMats_Parameters);

//permission controller to ensure that network ist not heated up if ambient temperature is too high
Controller_OuterCapillaryTubeMats_Permission(fSetpointValue := fTargetTemperature_HNLT_Cooling-fOffset_OuterCapillaryTubeMats_Permission,
	fActualValue := ambientState.fOutsideTemperature,
	eMode := eCTRL_MODE_ACTIVE,
	stParams := Controller_OuterCapillaryTubeMats_Permission_Parameters);

//control hvfa storage
//set hysteresis parameters for two-point controllers in low temperature heating network

Controller_Buffer_HVFA_HNLT_HVFAUnloading_Parameters.fHysteresisRange := 2;
Controller_Buffer_HVFA_HNLT_HVFAUnloading_Parameters.tCtrlCycleTime := GlobalVariables.tCtrlCycleTime_MAIN;
Controller_Buffer_HVFA_HNLT_HVFAUnloading_Parameters.tTaskCycleTime := GlobalVariables.tTaskCycleTime_MAIN;

Controller_Buffer_HVFA_HNLT_HVFALoading_Parameters.fHysteresisRange := 4;
Controller_Buffer_HVFA_HNLT_HVFALoading_Parameters.tCtrlCycleTime := GlobalVariables.tCtrlCycleTime_MAIN;
Controller_Buffer_HVFA_HNLT_HVFALoading_Parameters.tTaskCycleTime := GlobalVariables.tTaskCycleTime_MAIN;

Controller_HVFA_HNLT_Recooling_Parameters.fHysteresisRange := 4;
Controller_HVFA_HNLT_Recooling_Parameters.tCtrlCycleTime := GlobalVariables.tCtrlCycleTime_MAIN;
Controller_HVFA_HNLT_Recooling_Parameters.tTaskCycleTime := GlobalVariables.tTaskCycleTime_MAIN;

Controller_HVFA_HNLT_HVFAUnloadingPermission_Parameters.fHysteresisRange := 4;
Controller_HVFA_HNLT_HVFAUnloadingPermission_Parameters.tCtrlCycleTime := GlobalVariables.tCtrlCycleTime_MAIN;
Controller_HVFA_HNLT_HVFAUnloadingPermission_Parameters.tTaskCycleTime := GlobalVariables.tTaskCycleTime_MAIN;

Controller_HVFA_HNLT_HVFALoadingPermission_Parameters.fHysteresisRange := 4;
Controller_HVFA_HNLT_HVFALoadingPermission_Parameters.tCtrlCycleTime := GlobalVariables.tCtrlCycleTime_MAIN;
Controller_HVFA_HNLT_HVFALoadingPermission_Parameters.tTaskCycleTime := GlobalVariables.tTaskCycleTime_MAIN;

//buffer storage asks HVFA_HNLT for unloading when buffer storage temperature falls below limit
Controller_Buffer_HVFA_HNLT_HVFAUnloading(fSetpointValue := fTargetTemperature_HNLT_Heating+fOffset_TargetTemperature_HVFA_HNLT_Heating,
	fActualValue := hnltState.fMidTemperature,
	eMode := eCTRL_MODE_ACTIVE,
	stParams := Controller_Buffer_HVFA_HNLT_HVFAUnloading_Parameters);
	
//buffer storage asks HVFA_HNLT for loading when buffer storage temperature rises above limit
Controller_Buffer_HVFA_HNLT_HVFALoading(fSetpointValue := hnltState.fMidTemperature,
	fActualValue := fTargetTemperature_HNLT_Cooling - fOffset_Buffer_HVFA_HNLT_HVFALoading,
	eMode := eCTRL_MODE_ACTIVE,
	stParams := Controller_Buffer_HVFA_HNLT_HVFALoading_Parameters);

//hvfa storage may only be unloaded when upper temperature is between limits for unloading
Controller_HVFA_HNLT_HVFAUnloadingPermission(fSetpointValue := hnltState.fLowerTemperature_ActiveStorage,
	fActualValue := fTargetTemperature_HNLT_Heating,
	eMode := eCTRL_MODE_ACTIVE,
	stParams := Controller_HVFA_HNLT_HVFAUnloadingPermission_Parameters);
	
//hvfa storage may only be loaded when lower temperature is between limits for loading
Controller_HVFA_HNLT_HVFALoadingPermission(fSetpointValue := fTargetTemperature_HNLT_Cooling - fOffset_HVFA_HNLT_HVFALoadingPermission,
	fActualValue := hnltState.fLowerTemperature_ActiveStorage,
	eMode := eCTRL_MODE_ACTIVE,
	stParams := Controller_HVFA_HNLT_HVFALoadingPermission_Parameters);

//enable hvfa recooling during low temperature times in summer months	
Controller_HVFA_HNLT_Recooling(fSetpointValue := hnltState.fLowerTemperature_ActiveStorage,
	fActualValue := fTargetTemperature_HNLT_Cooling-fOffset_HVFA_HNLT_Recooling,
	eMode := eCTRL_MODE_ACTIVE,
	stParams := Controller_HVFA_HNLT_Recooling_Parameters);
(*	
IF hnltCnLinkageControl.bHeatingMode THEN
	hnltControl.bSetStatusOn_HVFASystem := (Controller_HVFA_HNLT_HVFALoadingPermission.bOut AND Controller_Buffer_HVFA_HNLT_HVFALoading.bOut) OR (Controller_HVFA_HNLT_HVFAUnloadingPermission.bOut AND Controller_Buffer_HVFA_HNLT_HVFAUnloading.bOut);
	hnltControl.bLoading_HVFASystem := Controller_HVFA_HNLT_HVFALoadingPermission.bOut AND Controller_Buffer_HVFA_HNLT_HVFALoading.bOut;
	hnltControl.bSetStatusOn_OuterCapillaryTubeMats := Controller_OuterCapillaryTubeMats.bOut AND Controller_OuterCapillaryTubeMats_Permission.bOut;
ELSE
	hnltControl.bSetStatusOn_HVFASystem := ((Controller_HVFA_HNLT_HVFALoadingPermission.bOut AND Controller_Buffer_HVFA_HNLT_HVFALoading.bOut) OR (Controller_HVFA_HNLT_HVFAUnloadingPermission.bOut AND Controller_Buffer_HVFA_HNLT_HVFAUnloading.bOut)) OR (Controller_HVFA_HNLT_Recooling.bOut AND Controller_OuterCapillaryTubeMats_Permission.bOut);
	hnltControl.bLoading_HVFASystem := Controller_HVFA_HNLT_HVFALoadingPermission.bOut AND Controller_Buffer_HVFA_HNLT_HVFALoading.bOut;
	hnltControl.bSetStatusOn_OuterCapillaryTubeMats := (Controller_OuterCapillaryTubeMats.bOut AND Controller_OuterCapillaryTubeMats_Permission.bOut) OR (Controller_HVFA_HNLT_Recooling.bOut AND Controller_OuterCapillaryTubeMats_Permission.bOut);
END_IF
*)

IF Clock.stClockState.fHour > 6 AND Clock.stClockState.fHour < 22 THEN
	hnltControl.bSetStatusOn_HVFASystem := (Controller_HVFA_HNLT_HVFALoadingPermission.bOut AND Controller_Buffer_HVFA_HNLT_HVFALoading.bOut);
	hnltControl.bLoading_HVFASystem := Controller_HVFA_HNLT_HVFALoadingPermission.bOut AND Controller_Buffer_HVFA_HNLT_HVFALoading.bOut;
	hnltControl.bSetStatusOn_OuterCapillaryTubeMats := Controller_OuterCapillaryTubeMats.bOut;
ELSE
	hnltControl.bSetStatusOn_HVFASystem := Controller_HVFA_HNLT_Recooling.bOut ;
	hnltControl.bLoading_HVFASystem := FALSE;
	hnltControl.bSetStatusOn_OuterCapillaryTubeMats := Controller_HVFA_HNLT_Recooling.bOut OR Controller_OuterCapillaryTubeMats.bOut;
END_IF

// hnltControl.bSetStatusOn_OuterCapillaryTubeMats := Controller_OuterCapillaryTubeMats.bOut; AND Controller_OuterCapillaryTubeMats_Permission.bOut;
END_METHOD

METHOD ControlHnltCnLinkage : BOOL
VAR_INPUT
END_VAR
//set hysteresis parameters for hnlt cn linkage systems
fOffset_TargetTemperature_HeatPump := 0;
Controller_HeatPump_Parameters.fHysteresisRange := 4;
Controller_HeatPump_Parameters.tCtrlCycleTime := GlobalVariables.tCtrlCycleTime_MAIN;
Controller_HeatPump_Parameters.tTaskCycleTime := GlobalVariables.tTaskCycleTime_MAIN;

fOffset_TargetTemperature_HeatPump_Upper_CN_Permission := 4;
Controller_HeatPump_Permission_Upper_CN_Parameters.fHysteresisRange := 2;
Controller_HeatPump_Permission_Upper_CN_Parameters.tCtrlCycleTime := GlobalVariables.tCtrlCycleTime_MAIN;
Controller_HeatPump_Permission_Upper_CN_Parameters.tTaskCycleTime := GlobalVariables.tTaskCycleTime_MAIN;

fOffset_TargetTemperature_HeatPump_Lower_CN_Permission := 3;
Controller_HeatPump_Permission_Lower_CN_Parameters.fHysteresisRange := 4;
Controller_HeatPump_Permission_Lower_CN_Parameters.tCtrlCycleTime := GlobalVariables.tCtrlCycleTime_MAIN;
Controller_HeatPump_Permission_Lower_CN_Parameters.tTaskCycleTime := GlobalVariables.tTaskCycleTime_MAIN;
	
//control heat pump depending on heating demand in hnlt

Controller_HeatPump(fSetpointValue := fTargetTemperature_HNLT_Heating+fOffset_TargetTemperature_HeatPump,
	fActualValue := hnltState.fUpperTemperature,
	eMode := eCTRL_MODE_ACTIVE,
	stParams := Controller_HeatPump_Parameters);
	
Controller_HeatPump_Permission_Upper_CN(fSetpointValue := fTargetTemperature_CN+fOffset_TargetTemperature_HeatPump_Upper_CN_Permission,
	fActualValue := cnState.fUpperTemperature,
	eMode := eCTRL_MODE_ACTIVE,
	stParams := Controller_HeatPump_Permission_Lower_CN_Parameters);

Controller_HeatPump_Permission_Lower_CN(fSetpointValue := cnState.fMidTemperature,
	fActualValue := fTargetTemperature_CN-fOffset_TargetTemperature_HeatPump_Lower_CN_Permission,
	eMode := eCTRL_MODE_ACTIVE,
	stParams := Controller_HeatPump_Permission_Lower_CN_Parameters);
	
hnltCnLinkageControl.bSetStatusOn_HeatPump := Controller_HeatPump.bOut AND Controller_HeatPump_Permission_Lower_CN.bOut AND Controller_HeatPump_Permission_Upper_CN.bOut;
hnltCnLinkageControl.fTargetTemperature_ProductionHall := localDefaultParameters.fTargetTemperature_ProductionHall;

hnltCnLinkageControl.bSetStatusOn_InnerCapillaryTubeMats := TRUE;
hnltCnLinkageControl.bSetStatusOn_UnderfloorHeating := TRUE;
END_METHOD

METHOD SetState : BOOL
VAR_INPUT
END_VAR
localState.fTargetTemperature_HNHT_Heating := fTargetTemperature_HNHT_Heating;
localState.fTargetTemperature_HNHT_Cooling := fTargetTemperature_HNHT_Cooling;
localState.fTargetTemperature_HNLT_Heating := fTargetTemperature_HNLT_Heating;
localState.fTargetTemperature_HNLT_Cooling := fTargetTemperature_HNLT_Cooling;
localState.fTargetTemperature_CN := fTargetTemperature_CN;
localState.fTargetTemperature_ProductionHall := localDefaultParameters.fTargetTemperature_ProductionHall;

localState.aTemperatureLimits_HNHT := aTemperatureLimits_HNHT;
localState.aTemperatureLimits_HNLT := aTemperatureLimits_HNLT;
localState.aTemperatureLimits_CN := aTemperatureLimits_CN;
localState.bAlgorithmPermission_HNHT := HNHT_Check.bPermission;
localState.bAlgorithmPermission_HNLT := HNLT_Check.bPermission;
localState.bAlgorithmPermission_CN := CN_Check.bPermission;	

// localState.bHeatingMode state is set in AmbientControl

localState.fFeedTemperature_HNHT := fTargetTemperature_HNHT_Heating+localDefaultParameters.fOffset_FeedTemperature_HNHT;
localState.fFeedTemperature_HNLT_Heating := fTargetTemperature_HNLT_Heating+localDefaultParameters.fOffset_FeedTemperature_HNLT_Heating;
localState.fFeedTemperature_HNLT_Cooling := fTargetTemperature_HNLT_Cooling-localDefaultParameters.fOffset_FeedTemperature_HNLT_Cooling;
localState.fFeedTemperature_CN := fTargetTemperature_CN-localDefaultParameters.fOffset_FeedTemperature_CN;
END_METHOD

METHOD SetTemperatures : BOOL
VAR_INPUT
END_VAR
//set internal variables depending on prodution mode
IF localSetParameters.bProductionModeActivated THEN
	fTargetTemperature_CN := localDefaultParameters.fTargetTemperature_CN_ProductionMode;
	fTargetTemperature_HNLT_Heating := localDefaultParameters.fTargetTemperature_HNLT_Heating_ProductionMode;
	fTargetTemperature_HNLT_Cooling := localDefaultParameters.fTargetTemperature_HNLT_Cooling_ProductionMode;
	fTargetTemperature_HNHT_Heating := localDefaultParameters.fTargetTemperature_HNHT_Heating_ProductionMode;
	fTargetTemperature_HNHT_Cooling := localDefaultParameters.fTargetTemperature_HNHT_Cooling_ProductionMode;
	aTemperatureLimits_CN := localDefaultParameters.aTemperatureLimits_CN_ProductionMode;
	aTemperatureLimits_HNLT := localDefaultParameters.aTemperatureLimits_HNLT_ProductionMode;
	aTemperatureLimits_HNHT := localDefaultParameters.aTemperatureLimits_HNHT_ProductionMode;

ELSE
	fTargetTemperature_CN := localDefaultParameters.fTargetTemperature_CN;
	fTargetTemperature_HNLT_Heating := localDefaultParameters.fTargetTemperature_HNLT_Heating;
	fTargetTemperature_HNLT_Cooling := localDefaultParameters.fTargetTemperature_HNLT_Cooling;
	fTargetTemperature_HNHT_Heating := localDefaultParameters.fTargetTemperature_HNHT_Heating;
	fTargetTemperature_HNHT_Cooling := localDefaultParameters.fTargetTemperature_HNHT_Cooling;
	aTemperatureLimits_CN := localDefaultParameters.aTemperatureLimits_CN;
	aTemperatureLimits_HNLT := localDefaultParameters.aTemperatureLimits_HNLT;
	aTemperatureLimits_HNHT := localDefaultParameters.aTemperatureLimits_HNHT;
END_IF

//set feed temperatures
hnhtControl.fFeedTemperature := fTargetTemperature_HNHT_Heating+localDefaultParameters.fOffset_FeedTemperature_HNHT;
hnhtControl.fTargetTemperature := fTargetTemperature_HNHT_Heating;
hnltControl.fFeedTemperature_Heating := fTargetTemperature_HNLT_Heating+localDefaultParameters.fOffset_FeedTemperature_HNLT_Heating;
hnltControl.fFeedTemperature_Cooling := fTargetTemperature_HNLT_Cooling-localDefaultParameters.fOffset_FeedTemperature_HNLT_Cooling;
cnControl.fFeedTemperature := fTargetTemperature_CN-localDefaultParameters.fOffset_FeedTemperature_CN;
hnhtHnltLinkageControl.fFeedTemperature_HNHT := hnhtControl.fFeedTemperature;
hnhtHnltLinkageControl.fFeedTemperature_HNLT_Heating := hnltControl.fFeedTemperature_Heating;
hnhtHnltLinkageControl.fFeedTemperature_HNLT_Cooling := hnltControl.fFeedTemperature_Cooling;
hnltCnLinkageControl.fFeedTemperature_CN := cnControl.fFeedTemperature;
hnltCnLinkageControl.fFeedTemperature_HNLT_Heating := hnltControl.fFeedTemperature_Heating;
hnltCnLinkageControl.fFeedTemperature_HNLT_Cooling := hnltControl.fFeedTemperature_Cooling;

//set algorithm permission depending on production mode to control structs
CN_Check(fInput := cnState.fMidTemperature,
	fLowerLimit := aTemperatureLimits_CN[1],
	fUpperLimit := aTemperatureLimits_CN[2]);
cnControl.bAlgorithmPermission := CN_Check.bPermission;
	
HNLT_Check(fInput := hnltState.fMidTemperature,
	fLowerLimit := aTemperatureLimits_HNLT[1],
	fUpperLimit := aTemperatureLimits_HNLT[2]);
hnltControl.bAlgorithmPermission := HNLT_Check.bPermission;
	
HNHT_Check(fInput := hnhtState.fMidTemperature,
	fLowerLimit := aTemperatureLimits_HNHT[1],
	fUpperLimit := aTemperatureLimits_HNHT[2]);	
hnhtControl.bAlgorithmPermission := HNHT_Check.bPermission;
	
hnltCnLinkageControl.bAlgorithmPermission_CN := cnControl.bAlgorithmPermission;
hnltCnLinkageControl.bAlgorithmPermission_HNLT := hnltControl.bAlgorithmPermission;
hnhtHnltLinkageControl.bAlgorithmPermission_HNHT := hnhtControl.bAlgorithmPermission;
hnhtHnltLinkageControl.bAlgorithmPermission_HNLT := hnltControl.bAlgorithmPermission;
hnhtCnLinkageControl.bAlgorithmPermission_CN := cnControl.bAlgorithmPermission;
hnhtCnLinkageControl.bAlgorithmPermission_HNHT := hnhtControl.bAlgorithmPermission;
END_METHOD

END_FUNCTION_BLOCK

// ---- POUs/05 Thermal Networks/FB_CoolingNetwork.TcPOU
FUNCTION_BLOCK FB_CoolingNetwork
VAR_INPUT
	//control struct for cn
	controlAutomatic : ST_CoolingNetworkControl;	
END_VAR
VAR_OUTPUT
	{attribute 'OPC.UA.DA' := '1'}
	localState : ST_ThermalNetworkState;
END_VAR
VAR
	//systems
	BufferStorage : FB_BufferStorage;
	eChillerSystem : FB_eChillerSystem;
	HVFASystem : FB_HVFAStorageSystem;
	CentralMachineCoolingSystem : FB_CN_CentralMachineCooling;
	FlywheelMassStorageSystem : FB_FlywheelMassStorageSystem;
	
	//machines
	EMAG_GT : FB_EMAG_GT;
	EMAG_Y : FB_EMAG_Y;
	FlyhweelMassStorage : FB_FlywheelMassStorage;
	
	//internal variables
	bSetStatusOn_CentralMachineCooling : BOOL;
	bSetStatusOn_FlywheelMassStorage : BOOL;
END_VAR

//buffer storage system
BufferStorage();
localState.fUpperTemperature := BufferStorage.localState.fUpperTemperature;
localState.fMidTemperature := BufferStorage.localState.fMidTemperature;
localState.fLowerTemperature := BufferStorage.localState.fLowerTemperature;
localState.fUpperTemperature_ActiveStorage := HVFASystem.localStorageState.fUpperTemperature;
localState.fLowerTemperature_ActiveStorage := HVFASystem.localStorageState.fLowerTemperature;

//machines
EMAG_Y();
bSetStatusOn_CentralMachineCooling := EMAG_Y.bCN_Demand;

FlyhweelMassStorage();
bSetStatusOn_FlywheelMassStorage := FlyhweelMassStorage.bStatusOn;

//producer
eChillerSystem(bSetStatusOnAutomatic := controlAutomatic.bSetStatusOn_eChiller,
	bAlgorithmPermission := controlAutomatic.bAlgorithmPermission,
	fSetPointAutomatic := controlAutomatic.fFeedTemperature,
	fExternalTemperature := BufferStorage.localState.fMidTemperature,
	fReturnTemperature_Consumers := BufferStorage.localState.fUpperTemperature);

//consumer
//PU100 in central machine cooling system controls temperature difference of 3 K
CentralMachineCoolingSystem(bSetStatusOnAutomatic := bSetStatusOn_CentralMachineCooling,
	bAlgorithmPermission := controlAutomatic.bAlgorithmPermission,
	fSetPointAutomatic := 3); //temperature difference control

//PU191 in central machine cooling system controls return temperature of 20 degree
FlywheelMassStorageSystem(bSetStatusOnAutomatic := bSetStatusOn_FlywheelMassStorage,
	bAlgorithmPermission := controlAutomatic.bAlgorithmPermission,
	fSetPointAutomatic := 3); //temperature difference control
	
//external storages
HVFASystem(bSetStatusOnAutomatic := controlAutomatic.bSetStatusOn_HVFASystem,
	bAlgorithmPermission := controlAutomatic.bAlgorithmPermission,
	fSetPointAutomatic := 40,
	bLoadingAutomatic := controlAutomatic.bLoading_HVFASystem,
	aTelegramm_WMZ7x0 := aTelegramm_WMZ710,
	aTelegramm_WMZx05 := aTelegramm_WMZ105);

END_FUNCTION_BLOCK

// ---- POUs/03 Storages/FB_BufferStorage.TcPOU
FUNCTION_BLOCK FB_BufferStorage
VAR_INPUT
END_VAR
VAR_OUTPUT
	{attribute 'OPC.UA.DA' := '1'}	
	localState : ST_BufferStorageState;
END_VAR
VAR
	UpperTemperatureSensor : FB_TemperatureSensor; //upper temperature sensor
	MidTemperatureSensor : FB_TemperatureSensor; //mid temperature sensor
	LowerTemperatureSensor : FB_TemperatureSensor; //lower temperature sensor
	PressureSensor : FB_PressureSensor; //pressure sensor
END_VAR

//sensors
UpperTemperatureSensor();
MidTemperatureSensor();
LowerTemperatureSensor();
PressureSensor();

//get sensor inputs
UpperTemperatureSensor.GetState_AI();
MidTemperatureSensor.GetState_AI();
LowerTemperatureSensor.GetState_AI();
PressureSensor.GetState_AI();

//set outputs
localState.fUpperTemperature := UpperTemperatureSensor.fTemperature;
localState.fMidTemperature := MidTemperatureSensor.fTemperature;
localState.fLowerTemperature := LowerTemperatureSensor.fTemperature;

END_FUNCTION_BLOCK

// ---- POUs/04 Systems/CoolingSystems/FB_eChillerSystem.TcPOU
FUNCTION_BLOCK FB_eChillerSystem EXTENDS FB_SystemContinous
VAR_INPUT
	fExternalTemperature : REAL; //External temperature of buffer storage
	fReturnTemperature_Consumers : REAL;
END_VAR
VAR_OUTPUT
END_VAR
VAR
	//Efficient Energy eChiller 45-II
	eChiller : FB_eChiller;
	
	//discrete valve 138
	stSV138DefaultParameters : ST_MixingValveDefaultParameters := (fControllerAmplification := 1, tControllerIntegralTime := T#100S, fOutMinLimit := 30,  tTaskCycleTime := GlobalVariables.tTaskCycleTime_MAIN, tCtrlCycleTime := GlobalVariables.tCtrlCycleTime_MAIN,fOffsetTerminal := 3950);
	SV138 : FB_MixingValve := (ST_DefaultParameters := stSV138DefaultParameters); //valve motor needs continous signal but operates only between extreme positions	
	
	//heat counters
	stWMZ135DefaultParameters : ST_MollineC3HeatCounterDefaultParameters := (fSpecificHeatCapacity := 4.7);
	WMZ135 : FB_MollineC3HeatCounter := (ST_DefaultParameters := stWMZ135DefaultParameters);
	WMZ138 : FB_MollineC3HeatCounter;
	EM138 : FB_EmonioP3;
	
	//internal variables
	bSetStatusOn_eChiller : BOOL;
	bSetStatusOn_SV138 : BOOL;
END_VAR

MAIN();
eChiller.GetState();
eChiller(
	bSetStatusOnAutomatic := bSetStatusOn_eChiller,
	fSetPointAutomatic := fSetPoint,
	bAlgorithmPermission := bAlgorithmPermission,
	fExternalTemperature := fExternalTemperature,
	fReturnTemperature_Consumers := fReturnTemperature_Consumers);
eChiller.SetState();

SV138.GetState_AI();
SV138(
	bSetStatusOnAutomatic := bSetStatusOn_SV138,
	fSetPointAutomatic := 100,
	bAlgorithmPermission := bAlgorithmPermission,
	fThermalPowerExternal := WMZ138.fHeatFlowRate,
	nControlModeAutomatic := 0);
SV138.SetState_AO();

//insert heat counter telegramm from other task
WMZ135(aHeatCounterTelegramm := aTelegramm_WMZ135);
WMZ138(aHeatCounterTelegramm := aTelegramm_WMZ138);
EM138(sIPAddr := GlobalVariables.sIP_Emonio_eChiller);

METHOD PROTECTED  CheckError : BOOL
VAR_INPUT
END_VAR
VAR
	bError_eChiller : BOOL := FALSE;
	bError_SV138 : BOOL := FALSE;
END_VAR
VAR_OUTPUT
	bError : BOOL := FALSE;
END_VAR
//check chiller for error
bError_eChiller := eChiller.bError;

//check valve SV138 for error
IF SV138.fOperatingPoint < 95 AND eChiller.bStatusOn THEN
	bError_SV138 := TRUE;
END_IF

bError := bError_eChiller OR bError_SV138;
END_METHOD

METHOD PROTECTED  Operational : BOOL
VAR_INPUT
END_VAR
VAR_OUTPUT
	bSwitchToWorking : BOOL := FALSE;
END_VAR
bSetStatusOn_eChiller := TRUE;

IF eChiller.bStatusOn THEN
	bSwitchToWorking := TRUE;
END_IF
END_METHOD

METHOD PROTECTED  RampDown : BOOL
VAR_INPUT
END_VAR
VAR_OUTPUT
	bRampDownFinished : BOOL := FALSE;
END_VAR
bSetStatusOn_eChiller := FALSE;

//wait until eChiller is switched off before closing valve
IF NOT eChiller.bStatusOn THEN
	bSetStatusOn_SV138 := FALSE;
	IF SV138.fOperatingPoint < 20  THEN
		bRampDownFinished := TRUE;
	END_IF
END_IF
END_METHOD

METHOD PROTECTED  RampUp : BOOL
VAR_INPUT
END_VAR
VAR_OUTPUT
	bRampUpFinished : BOOL := FALSE;
END_VAR
bSetStatusOn_SV138 := TRUE;

//wait until valve is opened
IF SV138.fOperatingPoint > 85 THEN
	bRampUpFinished := TRUE;
END_IF
END_METHOD

METHOD PROTECTED   SetSetPointLimits : BOOL
VAR_INPUT
END_VAR
aSetPointLimits[1] := eChiller.ST_DefaultParameters.aSetPointLimitsTemperature[1];
aSetPointLimits[2] := eChiller.ST_DefaultParameters.aSetPointLimitsTemperature[2];
END_METHOD

METHOD PROTECTED  SetState : BOOL
VAR_INPUT
END_VAR
VAR_OUTPUT
END_VAR
fOperatingPoint := fExternalTemperature;

controlState.bStatusOn := bSetStatusOn;
setPointState.aSetPointLimits := aSetPointLimits;
setPointState.fSetPoint := fSetPoint;
setPointState.fOperatingPoint := fOperatingPoint;
setPointState.sSetPointUnit := 'degreeC';
setPointState.sOperatingPointUnit := 'degreeC';
END_METHOD

METHOD PROTECTED  Working : BOOL
VAR_INPUT
END_VAR
VAR_OUTPUT
	bSwitchToOperational : BOOL := FALSE;
END_VAR
//empty method
END_METHOD

END_FUNCTION_BLOCK

// ---- POUs/01 Actuators/CoolingUnits/FB_eChiller.TcPOU
FUNCTION_BLOCK FB_eChiller EXTENDS FB_ActuatorContinous
VAR_INPUT
	fExternalTemperature : REAL;
	fReturnTemperature_Consumers : REAL;
END_VAR
VAR_OUTPUT
	bError : BOOL;
END_VAR
VAR
	//default parameters
	localDefaultParameters : ST_eChillerDefaultParameters;

	{attribute 'OPC.UA.DA' := '1'}
	localState : ST_eChillerState;
	
	//analog converters
	OutputConverter_SetpointValue : FB_AnalogOutput(fUpperLimit := 60, fLowerLimit := -30);
	OutputConverter_ActualTemperature : FB_AnalogOutput(fUpperLimit := 60, fLowerLimit := -30);
	OutputConverter_ReturnTemperature_Consumers : FB_AnalogOutput(fUpperLimit := 60, fLowerLimit := -30);
	
	//I/O Links
	nSetPoint_OUT						AT %Q* : INT;
	nActualTemperature_OUT 				AT %Q* : INT; //Actual temperature in buffer storage linked to terminal
	nReturnTemperature_Consumers_OUT 	AT %Q* : INT;
	bSetStatusOn_OUT 					AT %Q* : BOOL;
	bError_IN 							AT %I* : BOOL;
	bWarning_IN 						AT %I* : BOOL;
	bStatusOn_IN 						AT %I* : BOOL;
END_VAR

MAIN();
OutputConverter_SetpointValue(fValue := fSetPoint);
OutputConverter_ActualTemperature(fValue := fExternalTemperature);
OutputConverter_ReturnTemperature_Consumers(fValue := fReturnTemperature_Consumers);

METHOD GetState : BOOL
VAR_INPUT
END_VAR
//control state
controlState.bStatusOn := bStatusOn_IN;
bStatusOn := bStatusOn_IN;

//setpoint state
setPointState.fOperatingPoint := fExternalTemperature;
setPointState.sOperatingPointUnit := 'degreeC';
fOperatingPoint := fExternalTemperature;

//local state
bError := bError_IN;
localState.bError := bError_IN;
localState.bWarning := bWarning_IN;
END_METHOD

METHOD PROTECTED  SetSetPointLimits : BOOL
VAR_INPUT
END_VAR
aSetPointLimits[1] := localDefaultParameters.aSetPointLimitsTemperature[1];
aSetPointLimits[2] := localDefaultParameters.aSetPointLimitsTemperature[2];
END_METHOD

METHOD SetState : BOOL
VAR_INPUT
END_VAR
//setpoint state
setPointState.fSetPoint := fSetPoint;
setPointState.sSetPointUnit := 'degreeC';
setPointState.aSetPointLimits := aSetPointLimits;

//outputs
nSetPoint_OUT := OutputConverter_SetpointValue.nValue;
nActualTemperature_OUT := OutputConverter_ActualTemperature.nValue;
nReturnTemperature_Consumers_OUT := OutputConverter_ReturnTemperature_Consumers.nValue;
bSetStatusOn_OUT := bSetStatusOn;
END_METHOD

PROPERTY ST_DefaultParameters : REFERENCE TO ST_eChillerDefaultParameters
GET
ST_DefaultParameters REF= localDefaultParameters;
END_GET
SET
localDefaultParameters := ST_DefaultParameters;
END_SET
END_PROPERTY

END_FUNCTION_BLOCK

// ---- POUs/04 Systems/StorageSystems/FB_HVFAStorageSystem.TcPOU
FUNCTION_BLOCK FB_HVFAStorageSystem EXTENDS FB_SystemContinous
VAR_INPUT
	bLoadingAutomatic : BOOL; //variable to determine if storage is in loading mode
	aTelegramm_WMZ7x0 : ARRAY[1..cMBUS_MaxTelegrams] OF ST_MBus_Data2;
	aTelegramm_WMZx05 : ARRAY[1..cMBUS_MaxTelegrams] OF ST_MBus_Data2;
END_VAR
VAR_OUTPUT	
	localStorageState : ST_HVFAStorageState;
END_VAR
VAR
	{attribute 'OPC.UA.DA' := '1'}
	localSetParameters : ST_ActiveStorageSystemSetParameters;
	{attribute 'OPC.UA.DA' := '1'}
	localState : ST_ActiveStorageSystemState;
	
	//default parameters
	localDefaultParameters : ST_HVFAStorageSystemDefaultParameters;	

	//storage
	HVFAStorage : FB_HVFAStorage;
	
	//pumps
	PUx05 : FB_PumpGrundfosMagna3; //Magna 3 pump (network side)
	PU7x0 : FB_Pump2Point; //CM pump (storage side)

	//valves
	stSVx05DefaultParameters : ST_MixingValveDefaultParameters := (tTaskCycleTime := GlobalVariables.tCtrlCycleTime_MAIN, tCtrlCycleTime := GlobalVariables.tCtrlCycleTime_MAIN, fOffsetTerminal := 3950);
	stSVx06DefaultParameters : ST_MixingValveDefaultParameters := (tTaskCycleTime := GlobalVariables.tCtrlCycleTime_MAIN, tCtrlCycleTime := GlobalVariables.tCtrlCycleTime_MAIN, fOffsetTerminal := 3950);
	stRVx05DefaultParameters : ST_MixingValveDefaultParameters := (tTaskCycleTime := GlobalVariables.tCtrlCycleTime_MAIN, tCtrlCycleTime := GlobalVariables.tCtrlCycleTime_MAIN, fOffsetTerminal := 3950, fControllerAmplification := 0.01);
	
	SVx05 : FB_MixingValve := (ST_DefaultParameters := stSVx05DefaultParameters); //discrete inlet valve, valve motor needs continous signal but operates only between extreme positions
	SVx06 : FB_MixingValve := (ST_DefaultParameters := stSVx06DefaultParameters); //discrete outlet valve	, valve motor needs continous signal but operates only between extreme positions
	RVx05 : FB_MixingValve := (ST_DefaultParameters := stRVx05DefaultParameters); //continous mixing valve
	
	//sensors
	WMZ7x0 : FB_MollineC3HeatCounter;
	WMZx05 : FB_MollineC3HeatCounter;
	
	//internal variables
	bSetStatusOn_PUx05 : BOOL;
	bSetStatusOn_PU7x0 : BOOL;
	bSetStatusOn_SVx05 : BOOL;
	fSetPoint_SVx05 : REAL;
	bSetStatusOn_SVx06 : BOOL;
	fSetPoint_SVx06 : REAL;	
	bSetStatusOn_RVx05 : BOOL;
	bLoading : BOOL;
	
	//triggers
	SwitchToLoading : R_TRIG;
	SwitchToUnloading : F_TRIG;
	bFinishedSwitchMode : BOOL := TRUE;
END_VAR

//storage
HVFAStorage(localState => localStorageState);

SelectLocalControlMode();
SwitchToLoading(CLK := bLoading);
SwitchToUnloading(CLK := bLoading);

//MAIN must be called before SwitchMode to prevent pump signal chattering (signal is written after SwitchMode function), SwitchMode may only be called if system is on
MAIN();

//disrupt calling SystemFlowControl via MAIN() when mode is switched and call SwitchMode()
IF ((SwitchToLoading.Q OR SwitchToUnloading.Q) OR NOT bFinishedSwitchMode) AND bSetStatusOn THEN
	SwitchMode(bSwitchToLoading := bLoading,
		bFinishedSwitchMode => bFinishedSwitchMode);
END_IF;

//pumps
PUx05.GetState_Profibus();
PUx05(bSetStatusOnAutomatic := bSetStatusOn_PUx05,
	fSetPointAutomatic := fSetPoint,
	bAlgorithmPermission := bAlgorithmPermission,
	nControlModeAutomatic := 0);
PUx05.SetState_Profibus();

PU7x0(bSetStatusOnAutomatic := bSetStatusOn_PU7x0,
	bAlgorithmPermission := bAlgorithmPermission);
PU7x0.SetState_BO();

//valves
SVx05.GetState_AI();
SVx05(bSetStatusOnAutomatic := bSetStatusOn_SVx05,
	fSetPointAutomatic := fSetPoint_SVx05,
	bAlgorithmPermission := bAlgorithmPermission,
	nControlModeAutomatic := 0);
SVx05.SetState_AO();

SVx06.GetState_AI();
SVx06(bSetStatusOnAutomatic := bSetStatusOn_SVx06,
	fSetPointAutomatic := fSetPoint_SVx06,
	bAlgorithmPermission := bAlgorithmPermission,
	nControlModeAutomatic := 0);
SVx06.SetState_AO();

//insert heat counter telegramm from other task
WMZ7x0(aHeatCounterTelegramm := aTelegramm_WMZ7x0);
WMZx05(aHeatCounterTelegramm := aTelegramm_WMZx05);

RVx05.GetState_AI();
RVx05(bSetStatusOnAutomatic := bSetStatusOn_RVx05,
	fSetPointAutomatic := 100,
	bAlgorithmPermission := bAlgorithmPermission,
	fThermalPowerExternal := WMZx05.fHeatFlowRate,
	nControlModeAutomatic := 0);
RVx05.SetState_AO();

METHOD PROTECTED  CheckError : BOOL
VAR_INPUT
END_VAR
VAR_OUTPUT
	bError : BOOL;
END_VAR
VAR
	bError_PUx05 : BOOL;
END_VAR
//check for pump error
bError_PUx05 := PUx05.bError;
END_METHOD

METHOD PROTECTED  Operational : BOOL
VAR_INPUT
END_VAR
VAR_OUTPUT
	bSwitchToWorking : BOOL := FALSE;
END_VAR
//storage pump
bSetStatusOn_PU7x0 := TRUE;

//network pump
bSetStatusOn_PUx05 := TRUE;

//temperature controlling valve
bSetStatusOn_RVx05 := TRUE;

IF PUx05.bStatusOn THEN
	bSwitchToWorking := TRUE;
END_IF
END_METHOD

METHOD PROTECTED  RampDown : BOOL
VAR_INPUT
END_VAR
VAR_OUTPUT
	bRampDownFinished : BOOL := FALSE;
END_VAR
bSetStatusOn_PU7x0 := FALSE;
bSetStatusOn_PUx05 := FALSE;
bSetStatusOn_RVx05 := FALSE;

IF RVx05.fOperatingPoint<20 AND NOT PUx05.bStatusOn THEN
	bRampDownFinished := TRUE;
END_IF
END_METHOD

METHOD PROTECTED  RampUp : BOOL
VAR_INPUT
END_VAR
VAR_OUTPUT
	bRampUpFinished : BOOL := FALSE;
END_VAR
bSetStatusOn_SVx05 := TRUE;
bSetStatusOn_SVx06 := TRUE;

IF bLoading = TRUE THEN
	fSetPoint_SVx05 := 0;
	fSetPoint_SVx06 := 0;
	IF SVx05.fOperatingPoint<20 AND SVx06.fOperatingPoint<20 THEN
		bRampUpFinished := TRUE;
	END_IF
ELSE
	fSetPoint_SVx05 := 100;
	fSetPoint_SVx06 := 100;
	IF SVx05.fOperatingPoint>80 AND SVx06.fOperatingPoint>80 THEN
		bRampUpFinished := TRUE;
	END_IF
END_IF
END_METHOD

METHOD PRIVATE SelectLocalControlMode : BOOL
VAR_INPUT
END_VAR
IF control.bManualModeActivated THEN
	bLoading := localSetParameters.bLoadingManual;
ELSIF control.bAlgorithmModeActivated AND bAlgorithmPermission THEN
	bLoading := localSetParameters.bLoadingAlgorithm;
ELSE
	bLoading := bLoadingAutomatic;
END_IF
END_METHOD

METHOD PROTECTED   SetSetPointLimits : BOOL
VAR_INPUT
END_VAR
aSetPointLimits[1] := localDefaultParameters.aSetPointLimitsTemperature[1];
aSetPointLimits[2] := localDefaultParameters.aSetPointLimitsTemperature[2];
END_METHOD

METHOD PROTECTED  SetState : BOOL
VAR_INPUT
END_VAR
VAR_OUTPUT
END_VAR
fOperatingPoint := PUx05.fOperatingPoint;

IF SVx05.fOperatingPoint<20 AND SVx06.fOperatingPoint<20 THEN
	localState.bLoading := TRUE;
ELSE
	localState.bLoading := FALSE;
END_IF

controlState.bStatusOn := bSetStatusOn;
setPointState.aSetPointLimits := aSetPointLimits;
setPointState.fSetPoint := fSetPoint;
setPointState.fOperatingPoint := fOperatingPoint;
setPointState.sSetPointUnit := 'percent';
setPointState.sOperatingPointUnit := 'percent';
END_METHOD

PROPERTY ST_DefaultParameters : REFERENCE TO ST_HVFAStorageSystemDefaultParameters
SET
localDefaultParameters := ST_DefaultParameters;
END_SET
END_PROPERTY

METHOD PRIVATE SwitchMode : BOOL
VAR_INPUT
	bSwitchToLoading : BOOL; //if false switch to cooling
END_VAR
VAR_OUTPUT
	bFinishedSwitchMode : BOOL := FALSE;
END_VAR
VAR_INST
	bRampDownFinished : BOOL := FALSE;
END_VAR
//check system state
IF bRampDownFinished THEN
	IF bSwitchToLoading THEN
		fSetPoint_SVx05 := 0;
		fSetPoint_SVx06 := 0;
		IF SVx05.fOperatingPoint<20 AND SVx06.fOperatingPoint<20 THEN
			//reset instant variable and switch on pump
			bRampDownFinished := FALSE;			
			bFinishedSwitchMode := TRUE;
			bSetStatusOn_PUx05 := TRUE;
		END_IF
		
	ELSE
		fSetPoint_SVx05 := 100;
		fSetPoint_SVx06 := 100;
		IF SVx05.fOperatingPoint>80 AND SVx06.fOperatingPoint>80 THEN
			//reset instant variable and switch on pump
			bRampDownFinished := FALSE;			
			bFinishedSwitchMode := TRUE;
			bSetStatusOn_PUx05 := TRUE;
		END_IF
	END_IF
ELSE
	bSetStatusOn_PUx05 := FALSE;
	IF NOT PUx05.bStatusOn THEN
		bRampDownFinished := TRUE;
	END_IF
END_IF
END_METHOD

METHOD PROTECTED  Working : BOOL
VAR_INPUT
END_VAR
VAR_OUTPUT
	bSwitchToOperational : BOOL := FALSE;
END_VAR
//empty method
END_METHOD

END_FUNCTION_BLOCK

// ---- POUs/03 Storages/FB_HVFAStorage.TcPOU
FUNCTION_BLOCK FB_HVFAStorage
VAR_INPUT
END_VAR
VAR_OUTPUT
	{attribute 'OPC.UA.DA' := '1'}
	localState : ST_HVFAStorageState;
END_VAR
VAR
	UpperTemperatureSensor : FB_TemperatureSensor; //upper temperature sensor
	LowerTemperatureSensor : FB_TemperatureSensor; //lower temperature sensor
END_VAR

//get sensor inputs
UpperTemperatureSensor.GetState_AI();
LowerTemperatureSensor.GetState_AI();

//set outputs
localState.fUpperTemperature := UpperTemperatureSensor.fTemperature;
localState.fLowerTemperature := LowerTemperatureSensor.fTemperature;

END_FUNCTION_BLOCK

// ---- POUs/01 Actuators/Pumps/FB_Pump2Point.TcPOU
FUNCTION_BLOCK FB_Pump2Point EXTENDS FB_Actuator2Point
VAR
	//I/O Links
	bSetStatusOn_OUT 	AT %Q* : BOOL := FALSE;
END_VAR

SelectControlMode();

METHOD SetState_BO : BOOL
VAR_INPUT
END_VAR
//output
bSetStatusOn_OUT := bSetStatusOn;
END_METHOD

END_FUNCTION_BLOCK

// ---- POUs/04 Systems/ConsumerSystems/CN/FB_CN_CentralMachineCooling.TcPOU
FUNCTION_BLOCK FB_CN_CentralMachineCooling EXTENDS FB_SystemContinous
VAR_INPUT
END_VAR
VAR_OUTPUT
END_VAR
VAR
	//default parameters
	localDefaultParameters : ST_CN_CentralMachineCoolingDefaultParameters;
	
	//pumps
	stPU100DefaultParameters : ST_PumpGrundfosMagna3DefaultParameters := (tTaskCycleTime := GlobalVariables.tTaskCycleTime_MAIN, tCtrlCycleTime := GlobalVariables.tCtrlCycleTime_MAIN);
	PU100 : FB_PumpGrundfosMagna3 := (ST_DefaultParameters := stPU100DefaultParameters);;

	//valves
	stSV100DefaultParameters : ST_DiscreteValveDefaultParameters := (nFeedback := 3);
	SV100 : FB_DiscreteValve := (ST_DefaultParameters := stSV100DefaultParameters);
	
	//heat counters
	WMZ100: FB_MollineEHeatCounter;
	
	//internal variables
	bSetStatusOn_PU100 : BOOL;
	bSetStatusOn_SV100 : BOOL;
END_VAR

MAIN();

SV100.GetState_BI();
SV100(bSetStatusOnAutomatic := bSetStatusOn_SV100,
	bAlgorithmPermission := bAlgorithmPermission);
SV100.SetState_BO();

PU100.GetState_Profibus();
PU100(bSetStatusOnAutomatic := bSetStatusOn_PU100,
	bAlgorithmPermission := bAlgorithmPermission,
	fSetPointAutomatic := fSetPoint,
	nControlModeAutomatic := 3,
	fThermalPowerExternal := WMZ100.fHeatFlowRate);
PU100.SetState_Profibus();

WMZ100(aHeatCounterTelegramm:=aTelegramm_WMZ100);

METHOD PROTECTED  CheckError : BOOL
VAR_INPUT
END_VAR
VAR_OUTPUT
	bError : BOOL;
END_VAR
IF (PU100.bStatusOn AND SV100.localState.nPosition = 2) OR PU100.bError THEN
	bError := TRUE;
END_IF
END_METHOD

METHOD PROTECTED  Operational : BOOL
VAR_INPUT
END_VAR
VAR_OUTPUT
	bSwitchToWorking : BOOL := FALSE;
END_VAR
bSetStatusOn_PU100 := TRUE;

IF PU100.bStatusOn THEN
	bSwitchToWorking := TRUE;
END_IF
END_METHOD

METHOD PROTECTED  RampDown : BOOL
VAR_INPUT
END_VAR
VAR_OUTPUT
	bRampDownFinished : BOOL := FALSE;
END_VAR
bSetStatusOn_PU100 := FALSE;

IF NOT PU100.bStatusOn THEN
	bSetStatusOn_SV100 := FALSE;
	IF SV100.localState.nPosition = 2 THEN
		bRampDownFinished := TRUE;
	END_IF
END_IF
END_METHOD

METHOD PROTECTED  RampUp : BOOL
VAR_INPUT
END_VAR
VAR_OUTPUT
	bRampUpFinished : BOOL := FALSE;
END_VAR
bSetStatusOn_SV100 := TRUE;

IF SV100.localState.nPosition = 3 THEN
	bRampUpFinished := TRUE;
END_IF
END_METHOD

METHOD PROTECTED   SetSetPointLimits : BOOL
VAR_INPUT
END_VAR
IF  PU100.nControlModeAutomatic = 3 THEN
	aSetPointLimits[1] := localDefaultParameters.aSetPointLimitsTemperatureDifference[1];
	aSetPointLimits[2] := localDefaultParameters.aSetPointLimitsTemperatureDifference[2];
ELSE
	aSetPointLimits[1] := localDefaultParameters.aSetPointLimitsRelativeSpeed[1];
	aSetPointLimits[2] := localDefaultParameters.aSetPointLimitsRelativeSpeed[2];
END_IF
END_METHOD

METHOD PROTECTED  SetState : BOOL
VAR_INPUT
END_VAR
VAR_OUTPUT
END_VAR
fOperatingPoint := PU100.localState.fTemperatureDifference;

controlState.bStatusOn := bSetStatusOn;
setPointState.aSetPointLimits := aSetPointLimits;
setPointState.fSetPoint := fSetPoint;
setPointState.fOperatingPoint := fOperatingPoint;
setPointState.sSetPointUnit := 'K';
setPointState.sOperatingPointUnit := 'K';
END_METHOD

METHOD PROTECTED  Working : BOOL
VAR_INPUT
END_VAR
VAR_OUTPUT
	bSwitchToOperational : BOOL := FALSE;
END_VAR
//empty method
END_METHOD

END_FUNCTION_BLOCK

// ---- POUs/04 Systems/ConsumerSystems/CN/FB_FlywheelMassStorageSystem.TcPOU
FUNCTION_BLOCK FB_FlywheelMassStorageSystem EXTENDS FB_SystemContinous
VAR_INPUT
END_VAR
VAR_OUTPUT
END_VAR
VAR
	//default parameters
	localDefaultParameters : ST_FlywheelMassStorageDefaultParameters;	

	//pumps
	stPU191DefaultParameters : ST_PumpGrundfosMagna3DefaultParameters := (tTaskCycleTime := GlobalVariables.tTaskCycleTime_MAIN, tCtrlCycleTime := GlobalVariables.tCtrlCycleTime_MAIN);
	PU191 : FB_PumpGrundfosMagna3 := (ST_DefaultParameters := stPU191DefaultParameters);;

	//valves
	stSV191DefaultParameters : ST_DiscreteValveDefaultParameters := (nFeedback := 0);
	SV191 : FB_DiscreteValve := (ST_DefaultParameters := stSV191DefaultParameters);
	
	//internal variables
	bSetStatusOn_PU191 : BOOL;
	bSetStatusOn_SV191 : BOOL;
	
	bStartTimer : BOOL;
	Timer : TON;
END_VAR

MAIN();

//use timer because valve has no feedback signal
Timer(IN := bStartTimer,
	PT := T#75S);

SV191.GetState_BI();
SV191(bSetStatusOnAutomatic := bSetStatusOn_SV191,
	bAlgorithmPermission := bAlgorithmPermission);
SV191.SetState_BO();

//pump controls return temperature
PU191.GetState_Profibus();
PU191(bSetStatusOnAutomatic := bSetStatusOn_PU191,
	bAlgorithmPermission := bAlgorithmPermission,
	fSetPointAutomatic := fSetPoint,
	nControlModeAutomatic := 3);
PU191.SetState_Profibus();

METHOD PROTECTED  CheckError : BOOL
VAR_INPUT
END_VAR
VAR_OUTPUT
	bError : BOOL;
END_VAR
bError := PU191.bError;
END_METHOD

METHOD PROTECTED  Operational : BOOL
VAR_INPUT
END_VAR
VAR_OUTPUT
	bSwitchToWorking : BOOL := FALSE;
END_VAR
bSetStatusOn_PU191 := TRUE;

IF PU191.bStatusOn THEN
	bSwitchToWorking := TRUE;
END_IF
END_METHOD

METHOD PROTECTED  RampDown : BOOL
VAR_INPUT
END_VAR
VAR_OUTPUT
	bRampDownFinished : BOOL := FALSE;
END_VAR
bSetStatusOn_PU191 := FALSE;

IF NOT PU191.bStatusOn THEN
	bSetStatusOn_SV191 := FALSE;
	bStartTimer := TRUE;
	IF Timer.Q THEN
		bStartTimer := FALSE;
		bRampDownFinished := TRUE;
	END_IF
END_IF
END_METHOD

METHOD PROTECTED  RampUp : BOOL
VAR_INPUT
END_VAR
VAR_OUTPUT
	bRampUpFinished : BOOL := FALSE;
END_VAR
bSetStatusOn_SV191 := TRUE;
bStartTimer := TRUE;

IF Timer.Q THEN
	bStartTimer := FALSE;
	bRampUpFinished := TRUE;
END_IF
END_METHOD

METHOD PROTECTED   SetSetPointLimits : BOOL
VAR_INPUT
END_VAR
IF  PU191.nControlModeAutomatic = 3 THEN
	aSetPointLimits[1] := localDefaultParameters.aSetPointLimitsTemperatureDifference[1];
	aSetPointLimits[2] := localDefaultParameters.aSetPointLimitsTemperatureDifference[2];
ELSE
	aSetPointLimits[1] := localDefaultParameters.aSetPointLimitsRelativeSpeed[1];
	aSetPointLimits[2] := localDefaultParameters.aSetPointLimitsRelativeSpeed[2];
END_IF
END_METHOD

METHOD PROTECTED  SetState : BOOL
VAR_INPUT
END_VAR
VAR_OUTPUT
END_VAR
fOperatingPoint := PU191.localState.fTemperatureDifference;

controlState.bStatusOn := bSetStatusOn;
setPointState.aSetPointLimits := aSetPointLimits;
setPointState.fSetPoint := fSetPoint;
setPointState.fOperatingPoint := fOperatingPoint;
setPointState.sSetPointUnit := 'K';
setPointState.sOperatingPointUnit := 'K';
END_METHOD

METHOD PROTECTED  Working : BOOL
VAR_INPUT
END_VAR
VAR_OUTPUT
	bSwitchToOperational : BOOL := FALSE;
END_VAR
//empty method
END_METHOD

END_FUNCTION_BLOCK

// ---- POUs/01 Actuators/ConsumerUnits/FB_EMAG_GT.TcPOU
FUNCTION_BLOCK FB_EMAG_GT
VAR_INPUT
END_VAR
VAR_OUTPUT
	bStatusOn : BOOL;
	bError_Connection : BOOL;
END_VAR
VAR
	OPC_UA				: FB_OPC_UA_READ;
	stOPC_UA_Server		: ST_OPC_UA_Server;
	sOPC_UA_Server_URL 	: STRING;
	sNamespaceName		: STRING;
	aNodes				: ARRAY[1..2] OF ST_OPC_UANode;
	nNodeCount			: UDINT := 2;
	stIndexRange		: ARRAY [1..nMaxIndexRange] OF ST_UAIndexRange;
	currentNode			: UDINT := 1;
	
	bStatusOn_CoolingLubricant : BOOL;
	bStatusOn_Machine : BOOL;
	
	// timer
	bStartTimer : BOOL;
	Timer : TON;
END_VAR

sOPC_UA_Server_URL 	:= GlobalVariables.sIP_EMAG_GT;
sNamespaceName 		:= 'http://www.boschrexroth.com/IndraLogic';

(*Define Nodes to Read*)
aNodes[1].NodeID.sIdentifier			:= 'Application.Kuehlung_Anforderung.Kuehlung_KSS_blau_ON';
aNodes[1].NodeID.eIdentifierType		:= eUAIdentifierType_String;
aNodes[1].SizeOfDataType				:= DINT_TO_UDINT(eUAType_Boolean);
aNodes[1].NodeAddInfo.nIndexRangeCount 	:= 0;
aNodes[1].NodeAddInfo.stIndexRange		:= stIndexRange;
aNodes[1].TargetVar						:= ADR(bStatusOn_CoolingLubricant);

aNodes[2].NodeID.sIdentifier			:= 'Application.Kuehlung_Anforderung.Kuehlung_Maschine_blau_ON';
aNodes[2].NodeID.eIdentifierType		:= eUAIdentifierType_String;
aNodes[2].SizeOfDataType				:= DINT_TO_UDINT(eUAType_Boolean);
aNodes[2].NodeAddInfo.nIndexRangeCount 	:= 0;
aNodes[2].NodeAddInfo.stIndexRange		:= stIndexRange;
aNodes[2].TargetVar						:= ADR(bStatusOn_Machine);
bError_Connection := OPC_UA.bError_Connection;
Timer(IN := bStartTimer,
	PT := T#5S);

bStartTimer := TRUE;
IF Timer.Q THEN
	OPC_UA(
		stNode				:= aNodes[currentNode],
		sOPC_UA_Server_Url 	:= sOPC_UA_Server_URL,
		sNamespaceName		:= sNamespaceName);
	currentNode := currentNode + 1;
	IF currentNode > nNodeCount THEN
		currentNode := 1;
	END_IF
	bStartTimer := FALSE;
END_IF

bStatusOn := bStatusOn_CoolingLubricant OR bStatusOn_Machine;

END_FUNCTION_BLOCK

// ---- POUs/07 Utilities/FB_OPC_UA_Read.TcPOU
FUNCTION_BLOCK FB_OPC_UA_Read
VAR_INPUT
	stNode				: ST_OPC_UANode;
	sOPC_UA_Server_Url 	: STRING;
	sNamespaceName		: STRING;
END_VAR
VAR_OUTPUT
	bError_Connection : BOOL := FALSE;
END_VAR
VAR
	Node : ST_OPC_UANode;
	bError		: BOOL;
	iState		: INT 	:= 0;
	bBusy		: BOOL;
	nErrorID	: DWORD;

	SessionConnectInfo		: ST_UASessionConnectInfo;
	sOpcUA_URL				: STRING(MAX_STRING_LENGTH);
	nConnectionHdl			: DWORD;
	nNamespaceIndex			: UINT;

	fbUA_Connect			: UA_Connect;
	fbUA_GetNamespaceIndex	: UA_GetNamespaceIndex;
	fbUA_NodeGetHandle		: UA_NodeGetHandle;
	fbUA_Read				: UA_Read;
	fbUA_NodeReleaseHandle	: UA_NodeReleaseHandle;
	fbUA_Disconnect			: UA_Disconnect;

	stIndexRange			: ARRAY [1..nMaxIndexRange] OF ST_UAIndexRange;
	nIndexRangeCount		: UINT := 0;
END_VAR

CASE iState OF
	0: (* Start *)
		bError		:= FALSE;
		nErrorID	:= 0;

		(* Parameterize *)
		sOpcUA_URL						:= sOPC_UA_Server_Url;	(* OpcUA Url of the device with ip address *)

		SessionConnectInfo.tConnectTimeout 	:= T#1M;
		SessionConnectInfo.tSessionTimeout 	:= T#1M;
		SessionConnectInfo.sApplicationName	:= '';
		SessionConnectInfo.eSecurityMode 		:= eUASecurityMsgMode_None;
		SessionConnectInfo.eSecurityPolicyUri 	:= eUASecurityPolicy_None;
		SessionConnectInfo.eTransportProfileUri := eUATransportProfileUri_UATcp;

		stIndexRange[1].nStartIndex := 0;
		stIndexRange[1].nEndIndex := 1;
		Node := stNode;
		iState := iState + 1;

	1:	(* open UA session *)
		fbUA_Connect(
			Execute				:= TRUE,
			ServerURL			:= sOpcUA_URL,
			SessionConnectInfo	:= SessionConnectInfo,
			Timeout				:= T#5S,
			ConnectionHdl		=> nConnectionHdl
		);
		
		IF NOT fbUA_Connect.Busy THEN
			fbUA_Connect(Execute := FALSE);
	
			IF NOT fbUA_Connect.Error THEN
				(* session open *)
				iState := iState + 1;
				bError_Connection := FALSE;
			ELSE
				bError_Connection := TRUE;
				bError			:= TRUE;
				nErrorID		:= fbUA_Connect.ErrorID;
				nConnectionHdl	:= 0;
				iState 			:= 0;
			END_IF
		END_IF

		
	2:	(* Get Namespace Index *)

		fbUA_GetNamespaceIndex(
			Execute			:= TRUE,
			ConnectionHdl	:= nConnectionHdl,
			NamespaceUri	:= sNamespaceName,
			NamespaceIndex	=> Node.NodeID.nNamespaceIndex
		);


		IF NOT fbUA_GetNamespaceIndex.Busy THEN
			fbUA_GetNamespaceIndex(Execute := FALSE);
			IF NOT fbUA_GetNamespaceIndex.Error THEN
				iState		:= iState +1;
			ELSE
				bError		:= TRUE;
				nErrorID	:= fbUA_GetNamespaceIndex.ErrorID;
				iState 		:= 6;
			END_IF
		END_IF
	
	3:	(* Get Node Handle *)
		fbUA_NodeGetHandle(
			Execute			:= TRUE,
			ConnectionHdl	:= nConnectionHdl,
			NodeID			:= Node.NodeID,
			NodeHdl			=> Node.NodeHdl
		);

		IF NOT fbUA_NodeGetHandle.Busy THEN
			fbUA_NodeGetHandle(Execute := FALSE);
	
			IF NOT fbUA_NodeGetHandle.Error THEN
				iState		:= iState +1;
			ELSE
				bError		:= TRUE;
				nErrorID	:= fbUA_NodeGetHandle.ErrorID;
				iState 		:= 6;
			END_IF
		END_IF
	
	
	4: 	(* UA_Read *)
		fbUA_Read(
			Execute			:= TRUE,
			ConnectionHdl	:= nConnectionHdl,
			NodeHdl			:= Node.NodeHdl,
			cbData			:= Node.SizeOfDataType,
			stNodeAddInfo 	:= Node.NodeAddInfo,
			pVariable		:= Node.TargetVar
			);
	
		IF NOT fbUA_Read.Busy THEN
			fbUA_Read( Execute := FALSE);

			IF NOT fbUA_Read.Error THEN
				iState		:= iState+1;
			ELSE
				bError		:= TRUE;
				nErrorID	:= fbUA_Read.ErrorID;
				iState 		:= 6;
			END_IF
		END_IF


	5:	(* Release Node Handle *)
		fbUA_NodeReleaseHandle(
			Execute			:= TRUE,
			ConnectionHdl	:= nConnectionHdl,
			NodeHdl			:= Node.NodeHdl
		);

		IF NOT fbUA_NodeReleaseHandle.Busy THEN
			fbUA_NodeReleaseHandle(Execute := FALSE);

			IF  NOT fbUA_NodeReleaseHandle.Error THEN
				iState 		:= iState+1;
			ELSE
				bError		:= TRUE;
				nErrorID	:= fbUA_NodeReleaseHandle.ErrorID;
				iState 		:= 6;
			END_IF
		END_IF


	6:	(* close session *)
		fbUA_Disconnect(
			Execute			:= TRUE,
			ConnectionHdl	:= nConnectionHdl
		);
	
		IF NOT fbUA_Disconnect.Busy THEN
			fbUA_Disconnect(Execute := FALSE);
			bBusy := FALSE;
			IF NOT fbUA_Disconnect.Error THEN
				(* session closed *)
				iState 		:= 0;
			ELSE
				bError			:= TRUE;
				nErrorID		:= fbUA_Disconnect.ErrorID;
				iState 			:= 0;
				nConnectionHdl	:= 0;
			END_IF
		END_IF
END_CASE

END_FUNCTION_BLOCK

// ---- POUs/01 Actuators/ConsumerUnits/FB_EMAG_Y.TcPOU
FUNCTION_BLOCK FB_EMAG_Y
VAR_INPUT
	bCN_Demand : BOOL;
	bError_Connection : BOOL;
END_VAR
VAR_OUTPUT
END_VAR
VAR
	//I/O-Links
	Mode_IN AT %I* : BOOL;
	CoolingUnitOperational_IN AT %I* : BOOL;
	ConnectionStatus_IN AT %I* : BOOL;

END_VAR

bCN_Demand := CoolingUnitOperational_IN AND ConnectionStatus_IN;
bError_Connection := NOT ConnectionStatus_IN;

END_FUNCTION_BLOCK

// ---- POUs/01 Actuators/ConsumerUnits/FB_FlywheelMassStorage.TcPOU
FUNCTION_BLOCK FB_FlywheelMassStorage
VAR_OUTPUT
	bStatusOn : BOOL;
END_VAR
VAR
	OPC_UA				: FB_OPC_UA_READ;
	stOPC_UA_Server		: ST_OPC_UA_Server;
	sOPC_UA_Server_URL 	: STRING;
	sNamespaceName		: STRING;
	aNodes				: ARRAY[1..4] OF ST_OPC_UANode;
	nNodeCount			: UDINT := 4;
	stIndexRange		: ARRAY [1..nMaxIndexRange] OF ST_UAIndexRange;
	currentNode			: UDINT := 1;
END_VAR

sOPC_UA_Server_URL 	:= GlobalVariables.sIP_FlywheelMassStorage;
sNamespaceName 		:= 'http://www.boschrexroth.com/IndraLogic';

(*Define Nodes to Read*)
aNodes[1].NodeID.sIdentifier			:= 'Application.Elektrische_Energiespeicher.Zustand_Gesamt.Kuehlung_Anforderung';
aNodes[1].NodeID.eIdentifierType		:= eUAIdentifierType_String;
aNodes[1].SizeOfDataType				:= DINT_TO_UDINT(eUAType_Boolean);
aNodes[1].NodeAddInfo.nIndexRangeCount 	:= 0;
aNodes[1].NodeAddInfo.stIndexRange		:= stIndexRange;
aNodes[1].TargetVar						:= ADR(bStatusOn);

OPC_UA(
	stNode				:= aNodes[currentNode],
	sOPC_UA_Server_Url 	:= sOPC_UA_Server_URL,
	sNamespaceName		:= sNamespaceName);
currentNode := currentNode + 1;
IF currentNode > nNodeCount THEN
	currentNode := 1;
END_IF

END_FUNCTION_BLOCK

// ---- POUs/05 Thermal Networks/FB_HnltCnLinkage.TcPOU
FUNCTION_BLOCK FB_HnltCnLinkage
VAR_INPUT
	stAmbientState : ST_AmbientState;
	
	//control struct for hnlt cn linkage
	controlAutomatic : ST_HnltCnLinkageControl;
END_VAR
VAR_OUTPUT
END_VAR
VAR
	//systems
	HeatPumpSystem : FB_HeatPumpSystem_CN;
	InnerCapillaryTubeMats : FB_InnerCapillaryTubeMats;
	UnderfloorHeatingSystem : FB_UnderfloorHeatingSystem;
	
	//internal variables
	bAlgorithmPermission : BOOL;
END_VAR

//check for algorithm permission
bAlgorithmPermission := controlAutomatic.bAlgorithmPermission_CN AND controlAutomatic.bAlgorithmPermission_HNLT;
	
HeatPumpSystem(bSetStatusOnAutomatic := controlAutomatic.bSetStatusOn_HeatPump,
	bAlgorithmPermission := bAlgorithmPermission,
	fSetPointAutomatic := controlAutomatic.fFeedTemperature_HNLT_Heating);
	
//NOTE: inner capillary tube mats are always on and recieve desired hall temperature as setpoint
InnerCapillaryTubeMats(bSetStatusOnAutomatic := controlAutomatic.bSetStatusOn_InnerCapillaryTubeMats,
	bAlgorithmPermission := bAlgorithmPermission,
	fSetPointAutomatic := controlAutomatic.fTargetTemperature_ProductionHall,
	bHeatingModeAutomatic := controlAutomatic.bHeatingMode,
	stAmbientState := stAmbientState);

//NOTE: underfloor heating is always on and recieves no setpoint because ambient temperature depending feed temperature is calculated inside FB
UnderfloorHeatingSystem(bSetStatusOnAutomatic := controlAutomatic.bSetStatusOn_UnderfloorHeating,
	bAlgorithmPermission := bAlgorithmPermission,
	fSetPointAutomatic := 0,
	bHeatingModeAutomatic := controlAutomatic.bHeatingMode,
	stAmbientState := stAmbientState);

END_FUNCTION_BLOCK

// ---- POUs/04 Systems/LinkageSystems/FB_HeatPumpSystem_CN.TcPOU
FUNCTION_BLOCK FB_HeatPumpSystem_CN EXTENDS FB_SystemContinous
VAR_INPUT
END_VAR
VAR_OUTPUT
END_VAR
VAR
	//Vitocal 350-G heat pump
	HeatPump : FB_HeatPump;
	
	//valve 146 and valve 246
	ST_SV146DefaultParameters : ST_DiscreteValveDefaultParameters := (nFeedback := 0);
	ST_SV246DefaultParameters : ST_DiscreteValveDefaultParameters := (nFeedback := 0);	
	SV146 : FB_DiscreteValve := (ST_DefaultParameters := ST_SV146DefaultParameters);
	SV246 : FB_DiscreteValve := (ST_DefaultParameters := ST_SV246DefaultParameters);	
	
	//internal variables
	bSetStatusOn_HeatPump : BOOL;
	bSetStatusOn_SV146 : BOOL;
	bSetStatusOn_SV246 : BOOL;
	
	//sensors
	WMZ146 : FB_StarkMultical302HeatCounter;
	WMZ246 : FB_StarkMultical302HeatCounter;
	EM146 : FB_EmonioP3;
	
	bStartRampUpTimer : BOOL;
	bStartRampDownTimer : BOOL;
	RampUpTimer : TON;
	RampDownTimer : TON;
	
END_VAR

MAIN();
//use timer because valve has no feedback signal (75 sec)
RampUpTimer(IN := bStartRampUpTimer,
	PT := T#75S);

//use longer ramp down timer, because heat pump should be off before closing valves	
RampDownTimer(IN := bStartRampDownTimer,
	PT := T#240S);

//heat pump
HeatPump.GetState();
HeatPump(bSetStatusOnAutomatic := bSetStatusOn_HeatPump,
	bAlgorithmPermission := bAlgorithmPermission,
	fSetPointAutomatic := fSetPoint);
HeatPump.SetState();

//valves
SV146.GetState_BI();
SV146(bSetStatusOnAutomatic := bSetStatusOn_SV146,
		bAlgorithmPermission := bAlgorithmPermission);
SV146.SetState_BO();

SV246.GetState_BI();
SV246(bSetStatusOnAutomatic := bSetStatusOn_SV246,
		bAlgorithmPermission := bAlgorithmPermission);
SV246.SetState_BO();

//sensors
WMZ146(aHeatCounterTelegramm := Telegramm_WZ_4372_WP_946);
WMZ246(aHeatCounterTelegramm := Telegramm_WZ_4371_WP_946);
EM146(sIPAddr := GlobalVariables.sIP_Emonio_CN_HeatPump);

METHOD PROTECTED  CheckError : BOOL
VAR_INPUT
END_VAR
VAR_OUTPUT
	bError : BOOL;
END_VAR
//empty method because system has no feedback signals
END_METHOD

METHOD PROTECTED  Operational : BOOL
VAR_INPUT
END_VAR
VAR_OUTPUT
	bSwitchToWorking : BOOL := FALSE;
END_VAR
bSetStatusOn_HeatPump := TRUE;
bSwitchToWorking := TRUE;
END_METHOD

METHOD PROTECTED  RampDown : BOOL
VAR_INPUT
END_VAR
VAR_OUTPUT
	bRampDownFinished : BOOL := FALSE;
END_VAR
bSetStatusOn_HeatPump := FALSE;
bStartRampDownTimer := TRUE;

IF RampDownTimer.Q THEN
	bSetStatusOn_SV146 := FALSE;
	bSetStatusOn_SV246 := FALSE;
	bRampDownFinished := TRUE;
	bStartRampDownTimer := FALSE;
END_IF
END_METHOD

METHOD PROTECTED  RampUp : BOOL
VAR_INPUT
END_VAR
VAR_OUTPUT
	bRampUpFinished : BOOL := FALSE;
END_VAR
bSetStatusOn_SV146 := TRUE;
bSetStatusOn_SV246 := TRUE;
bStartRampUpTimer := TRUE;

IF RampUpTimer.Q THEN
	bRampUpFinished := TRUE;
	bStartRampUpTimer := FALSE; //resets timer
END_IF
END_METHOD

METHOD PROTECTED   SetSetPointLimits : BOOL
VAR_INPUT
END_VAR
//heat pump has no continous setpoint (limits are not used) but must be implemented because of abstract method
aSetPointLimits[1] := 0;
aSetPointLimits[2] := 100;
END_METHOD

METHOD PROTECTED  SetState : BOOL
VAR_INPUT
END_VAR
VAR_OUTPUT
END_VAR
fOperatingPoint := 0;

controlState.bStatusOn := bSetStatusOn;
setPointState.aSetPointLimits := aSetPointLimits;
setPointState.fSetPoint := 0;
setPointState.fOperatingPoint := fOperatingPoint;
setPointState.sSetPointUnit := '-';
setPointState.sOperatingPointUnit := '-';
END_METHOD

METHOD PROTECTED  Working : BOOL
VAR_INPUT
END_VAR
VAR_OUTPUT
	bSwitchToOperational : BOOL := FALSE;
END_VAR
//empty method because setpoint does not change during operation
END_METHOD

END_FUNCTION_BLOCK

// ---- POUs/01 Actuators/HeatingUnits/FB_HeatPump.TcPOU
FUNCTION_BLOCK FB_HeatPump EXTENDS FB_ActuatorContinous
VAR_INPUT
END_VAR
VAR_OUTPUT
	bError : BOOL;
END_VAR
VAR
	{attribute 'OPC.UA.DA' := '1'}
	localState : ST_HeatPumpState;
	
	//default parameters
	localDefaultParameters : ST_HeatPumpDefaultParameters;
	
	//analog converters
	OutputConverter : FB_AnalogOutput(fUpperLimit := 100, fLowerLimit := 0);
	
	//I/O Links
	nSetPoint_OUT			AT %Q* : INT;
	bSetStatusOn_OUT 		AT %Q* : BOOL;
	bStatusOn_IN			AT %I* : BOOL;
	bError_IN 				AT %I* : BOOL;
END_VAR

MAIN();
OutputConverter(fValue := fSetPoint);

METHOD GetState : BOOL
VAR_INPUT
END_VAR
//local state
controlState.bStatusOn := bStatusOn_IN;
localState.bError := bError_IN;
bStatusOn := controlState.bStatusOn;
bError := localState.bError;
END_METHOD

METHOD PROTECTED  SetSetPointLimits : BOOL
VAR_INPUT
END_VAR
aSetPointLimits[1] := localDefaultParameters.aSetPointLimitsTemperature[1];
aSetPointLimits[2] := localDefaultParameters.aSetPointLimitsTemperature[2];
END_METHOD

METHOD SetState : BOOL
VAR_INPUT
END_VAR
setPointState.fSetPoint := fSetPoint;
setPointState.aSetPointLimits := aSetPointLimits;
setPointState.sSetPointUnit := 'degreeC';

nSetPoint_OUT := OutputConverter.nValue;
bSetStatusOn_OUT := bSetStatusOn;
END_METHOD

PROPERTY ST_DefaultParameters : REFERENCE TO ST_HeatPumpDefaultParameters
GET
ST_DefaultParameters REF= localDefaultParameters;
END_GET
SET
localDefaultParameters := ST_DefaultParameters;
END_SET
END_PROPERTY

END_FUNCTION_BLOCK

// ---- POUs/04 Systems/LinkageSystems/FB_InnerCapillaryTubeMats.TcPOU
FUNCTION_BLOCK FB_InnerCapillaryTubeMats EXTENDS FB_SystemContinous
VAR_INPUT
	bHeatingModeAutomatic : BOOL; //control mode: 0 = heating mode, 1 = cooling mode
	stAmbientState : ST_AmbientState;
END_VAR
VAR_OUTPUT
END_VAR
VAR
	{attribute 'OPC.UA.DA' := '1'}
	localSetParameters : ST_InnerCapillaryTubeMatsSetParameters;

	//default parameters
	localDefaultParameters : ST_InnerCapillaryTubeMatsDefaultParameters;	
	
	//pumps
	stPU405DefaultParameters : ST_PumpGrundfosMagna3DefaultParameters;
	stPU500DefaultParameters : ST_PumpGrundfosMagna3DefaultParameters := (fMaximumVolumeFlowRate := 0.0083, fNominalVolumeFlowRate := 0.0019, fMaximumPressureDifference := 145000);
	
	PU405 : FB_PumpGrundfosMagna3 := (ST_DefaultParameters := stPU405DefaultParameters);
	PU500 : FB_PumpGrundfosMagna3 := (ST_DefaultParameters := stPU500DefaultParameters);	
	
	//valves
	stSV_CN_DefaultParameters : ST_DiscreteValveDefaultParameters := (nFeedback := 3);
	stSV_HNLT_DefaultParameters : ST_DiscreteValveDefaultParameters := (nFeedback := 3);
	stSV505DefaultParameters : ST_DiscreteValveDefaultParameters := (nFeedback := 3);
	stRV500DefaultParameters : ST_MixingValveDefaultParameters := (bFeedbackSignal := FALSE, tTaskCycleTime := GlobalVariables.tTaskCycleTime_MAIN, tCtrlCycleTime := GlobalVariables.tCtrlCycleTime_MAIN);	
	stRV5xxDefaultParameters : ST_MixingValveDefaultParameters := (bFeedbackSignal := FALSE, fControllerAmplification := 500, tControllerIntegralTime := T#240M, bARWOnIPartOnly := FALSE, tTaskCycleTime := GlobalVariables.tTaskCycleTime_MAIN, tCtrlCycleTime := GlobalVariables.tCtrlCycleTime_MAIN);
	
	SV_CN : FB_DiscreteValve := (ST_DefaultParameters := stSV_CN_DefaultParameters); //heating network supply
	SV_HNLT : FB_DiscreteValve := (ST_DefaultParameters := stSV_HNLT_DefaultParameters); //heating entwork return
	SV505 : FB_DiscreteValve := (ST_DefaultParameters := stSV505DefaultParameters); //PWT2
	RV500 : FB_MixingValve := (ST_DefaultParameters := stRV500DefaultParameters);
	RV541 : FB_MixingValve := (ST_DefaultParameters := stRV5xxDefaultParameters); //wall east 1
	RV542 : FB_MixingValve := (ST_DefaultParameters := stRV5xxDefaultParameters); //wall east 2
	RV543 : FB_MixingValve := (ST_DefaultParameters := stRV5xxDefaultParameters); //wall east 3
	RV551 : FB_MixingValve := (ST_DefaultParameters := stRV5xxDefaultParameters); //ceiling east 1
	RV552 : FB_MixingValve := (ST_DefaultParameters := stRV5xxDefaultParameters); //ceiling east 2
	RV553 : FB_MixingValve := (ST_DefaultParameters := stRV5xxDefaultParameters); //ceiling east 3
	RV561 : FB_MixingValve := (ST_DefaultParameters := stRV5xxDefaultParameters); //wall west 1
	RV562 : FB_MixingValve := (ST_DefaultParameters := stRV5xxDefaultParameters); //wall west 2
	RV563 : FB_MixingValve := (ST_DefaultParameters := stRV5xxDefaultParameters); //wall west 3
	RV571 : FB_MixingValve := (ST_DefaultParameters := stRV5xxDefaultParameters); //ceiling west 1
	RV572 : FB_MixingValve := (ST_DefaultParameters := stRV5xxDefaultParameters); //ceiling west 2
	RV573 : FB_MixingValve := (ST_DefaultParameters := stRV5xxDefaultParameters); //ceiling west 3
	
	//sensors
	PS500 : FB_PressureSensor;
	TS541 : FB_TemperatureSensor; //wall east section 1
	TS542 : FB_TemperatureSensor; //wall east section 2
	TS543 : FB_TemperatureSensor; //wall east section 3
	TS551 : FB_TemperatureSensor; //ceiling east section 1
	TS552 : FB_TemperatureSensor; //ceiling east section 2
	TS553 : FB_TemperatureSensor; //ceiling east section 3
	TS561 : FB_TemperatureSensor; //wall west section 1
	TS562 : FB_TemperatureSensor; //wall west section 2
	TS563 : FB_TemperatureSensor; //wall west section 3
	TS571 : FB_TemperatureSensor; //ceiling west section 1
	TS572 : FB_TemperatureSensor; //ceiling west section 2
	TS573 : FB_TemperatureSensor; //ceiling west section 3
	
	WMZ405 : FB_MollineEHeatCounter;
	
	//internal variables
	bHeatingMode 			: BOOL;
	bSetStatusOn_PU405 		: BOOL;
	bSetStatusOn_PU500 		: BOOL;
	bSetStatusOn_SV_HNLT	: BOOL;
	bSetStatusOn_SV_CN		: BOOL;
	bSetStatusOn_RV500 		: BOOL;
	fSetPoint_RV500 		: REAL;
	nControlMode_RV500 		: E_MixingValveControlMode; 	
	
	
	//characteristic curves and controllers
	CharacteristicCurve 			: FB_CTRL_FLOW_TEMP_SETPOINT_GEN;
	CharacteristicCurve_Parameters	: ST_CTRL_FLOW_TEMP_SETPOINT_GEN_PARAMS;
	
	//Moving Average
	Moving_Average_Hall_Temperature : FB_CTRL_MOVING_AVERAGE;
	fMeanHallTemperature : REAL;
	
	//triggers
	SwitchToHeating : R_TRIG;
	SwitchToCooling : F_TRIG;
	bFinishedSwitchMode : BOOL := TRUE;
	
	//clock
	stDefaultParameters_Clock : ST_ClockDefaultParameters := (tTaskCycleTime := GlobalVariables.tCtrlCycleTime_MAIN, tCtrlCycleTime := T#1M);
	Clock : FB_Clock := (ST_DefaultParameters := stDefaultParameters_Clock);
END_VAR

//check if heating mode has switched
SelectLocalControlMode();
LocalControl();
SwitchToHeating(CLK := bHeatingMode);
SwitchToCooling(CLK := bHeatingMode);

//MAIN must be called before SwitchMode to prevent pump signal chattering (signal is written after SwitchMode function), SwitchMode may only be called if system is on
MAIN();

//disrupt calling SystemFlowControl via MAIN() when mode is switched and call SwitchMode()
IF ((SwitchToHeating.Q OR SwitchToCooling.Q) OR NOT bFinishedSwitchMode) AND bSetStatusOn THEN
	SwitchMode(bSwitchToHeating := bHeatingMode,
		bFinishedSwitchMode => bFinishedSwitchMode);
END_IF;

//clock for night setback
Clock();

//pumps
PU405.GetState_Profibus();
PU405(bSetStatusOnAutomatic := bSetStatusOn_PU405,
	fSetPointAutomatic := 50,
	bAlgorithmPermission := bAlgorithmPermission,
	nControlModeAutomatic := 0);
PU405.SetState_Profibus();

PU500.GetState_Profibus();
PU500(bSetStatusOnAutomatic := bSetStatusOn_PU500,
	fSetPointAutomatic := 50,
	bAlgorithmPermission := bAlgorithmPermission,
	nControlModeAutomatic := 0);
PU500.SetState_Profibus();

//valves in thermal networks
RV500.GetState_AI();
RV500(bSetStatusOnAutomatic := bSetStatusOn_RV500,
	fSetPointAutomatic := fSetPoint_RV500,
	bAlgorithmPermission := bAlgorithmPermission,
	fTemperatureExternal := PU500.fTemperatureInternal,
	fThermalPowerExternal := WMZ405.fHeatFlowRate,
	nControlModeAutomatic := nControlMode_RV500);
RV500.SetState_AO();

SV_CN.GetState_BI();
SV_CN(bSetStatusOnAutomatic := bSetStatusOn_SV_CN,
	bAlgorithmPermission := bAlgorithmPermission);
SV_CN.SetState_BO();

SV_HNLT.GetState_BI();
SV_HNLT(bSetStatusOnAutomatic := bSetStatusOn_SV_HNLT,
	bAlgorithmPermission := bAlgorithmPermission);
SV_HNLT.SetState_BO();

//PWT2 is always closed
SV505.GetState_BI();
SV505(bSetStatusOnAutomatic := FALSE,
	bAlgorithmPermission := bAlgorithmPermission);
SV505.SetState_BO();

//Calculate Average Hall Temperature
CalculateAverageTemperature(fActualTemperature := stAmbientState.fHallTemperature, fMeanTemperature => fMeanHallTemperature);

//control valves in capillary tube mats
RV541.GetState_AI();
RV541(bSetStatusOnAutomatic := bSetStatusOn_RV500,
	fSetPointAutomatic := fSetPoint,
	bAlgorithmPermission := bAlgorithmPermission,
	fTemperatureExternal := fMeanHallTemperature,
	nControlModeAutomatic := nControlMode_RV500);
RV541.SetState_AO();

RV542.GetState_AI();
RV542(bSetStatusOnAutomatic := bSetStatusOn_RV500,
	fSetPointAutomatic := fSetPoint,
	bAlgorithmPermission := bAlgorithmPermission,
	fTemperatureExternal := fMeanHallTemperature,
	nControlModeAutomatic := nControlMode_RV500);
RV542.SetState_AO();

RV543.GetState_AI();
RV543(bSetStatusOnAutomatic := bSetStatusOn_RV500,
	fSetPointAutomatic := fSetPoint,
	bAlgorithmPermission := bAlgorithmPermission,
	fTemperatureExternal := fMeanHallTemperature,
	nControlModeAutomatic := nControlMode_RV500);
RV543.SetState_AO();

RV551.GetState_AI();
RV551(bSetStatusOnAutomatic := bSetStatusOn_RV500,
	fSetPointAutomatic := fSetPoint,
	bAlgorithmPermission := bAlgorithmPermission,
	fTemperatureExternal := fMeanHallTemperature,
	nControlModeAutomatic := nControlMode_RV500);
RV551.SetState_AO();

RV552.GetState_AI();
RV552(bSetStatusOnAutomatic := bSetStatusOn_RV500,
	fSetPointAutomatic := fSetPoint,
	bAlgorithmPermission := bAlgorithmPermission,
	fTemperatureExternal := fMeanHallTemperature,
	nControlModeAutomatic := nControlMode_RV500);
RV552.SetState_AO();

RV553.GetState_AI();
RV553(bSetStatusOnAutomatic := bSetStatusOn_RV500,
	fSetPointAutomatic := fSetPoint,
	bAlgorithmPermission := bAlgorithmPermission,
	fTemperatureExternal := fMeanHallTemperature,
	nControlModeAutomatic := nControlMode_RV500);
RV553.SetState_AO();

RV561.GetState_AI();
RV561(bSetStatusOnAutomatic := bSetStatusOn_RV500,
	fSetPointAutomatic := fSetPoint,
	bAlgorithmPermission := bAlgorithmPermission,
	fTemperatureExternal := fMeanHallTemperature,
	nControlModeAutomatic := nControlMode_RV500);
RV561.SetState_AO();

RV562.GetState_AI();
RV562(bSetStatusOnAutomatic := bSetStatusOn_RV500,
	fSetPointAutomatic := fSetPoint,
	bAlgorithmPermission := bAlgorithmPermission,
	fTemperatureExternal := fMeanHallTemperature,
	nControlModeAutomatic := nControlMode_RV500);
RV562.SetState_AO();

RV563.GetState_AI();
RV563(bSetStatusOnAutomatic := bSetStatusOn_RV500,
	fSetPointAutomatic := fSetPoint,
	bAlgorithmPermission := bAlgorithmPermission,
	fTemperatureExternal := fMeanHallTemperature,
	nControlModeAutomatic := nControlMode_RV500);
RV563.SetState_AO();

